C03636=1036.539,281.709,383.369,171.291,43.258,158.298
C03637=1036.532,281.461,383.400,171.287,43.257,158.298
C03638=1036.526,281.213,383.432,171.284,43.256,158.297
C03639=1036.519,280.965,383.463,171.280,43.255,158.297
C03640=1036.512,280.717,383.495,171.277,43.254,158.296
C03641=1036.506,280.468,383.525,171.273,43.253,158.295
C03642=1036.499,280.221,383.557,171.270,43.252,158.295
C03643=1036.492,279.973,383.588,171.266,43.251,158.294
C03644=1036.485,279.725,383.620,171.262,43.250,158.294
C03645=1036.479,279.477,383.651,171.259,43.249,158.293
C03646=1036.472,279.229,383.683,171.255,43.247,158.293
C03647=1036.465,278.981,383.714,171.252,43.247,158.292
C03648=1036.459,278.733,383.745,171.249,43.245,158.292
C03649=1036.452,278.485,383.776,171.245,43.244,158.291
C03650=1036.445,278.237,383.807,171.242,43.243,158.291
C03651=1036.438,277.989,383.838,171.238,43.242,158.290
C03652=1036.429,277.655,383.881,171.233,43.241,158.290
C03653=1036.420,277.319,383.922,171.229,43.240,158.289
C03654=1036.411,276.985,383.964,171.224,43.238,158.288
C03655=1036.401,276.651,384.006,171.219,43.237,158.288
C03656=1036.395,276.402,384.036,171.216,43.236,158.287
C03657=1036.388,276.154,384.068,171.212,43.235,158.287
C03658=1036.382,275.906,384.098,171.208,43.234,158.286
C03659=1036.374,275.658,384.129,171.205,43.233,158.286
C03660=1036.368,275.411,384.160,171.201,43.232,158.285
C03661=1036.362,275.162,384.191,171.198,43.231,158.285
C03662=1036.354,274.915,384.222,171.194,43.230,158.284
C03663=1036.348,274.666,384.253,171.191,43.229,158.284
C03664=1036.341,274.418,384.284,171.187,43.228,158.283
C03665=1036.335,274.170,384.315,171.185,43.227,158.283
C03666=1036.328,273.923,384.345,171.181,43.226,158.282
C03667=1036.321,273.674,384.376,171.177,43.225,158.282
C03668=1036.314,273.427,384.407,171.174,43.224,158.281
C03669=1036.308,273.178,384.438,171.170,43.223,158.281
C03670=1036.301,272.930,384.469,171.167,43.222,158.280
C03671=1036.294,272.682,384.499,171.163,43.222,158.280
C03672=1036.288,272.434,384.529,171.160,43.220,158.279
C03673=1036.280,272.187,384.560,171.156,43.220,158.279
C03674=1036.274,271.938,384.591,171.153,43.219,158.279
C03675=1036.267,271.690,384.622,171.150,43.217,158.278
C03676=1036.260,271.442,384.653,171.147,43.217,158.278
C03677=1036.254,271.194,384.683,171.143,43.216,158.277
C03678=1036.247,270.947,384.714,171.139,43.215,158.277
C03679=1036.240,270.698,384.744,171.136,43.214,158.276
C03680=1036.233,270.450,384.775,171.132,43.213,158.276
C03681=1036.227,270.202,384.805,171.129,43.212,158.275
C03682=1036.220,269.955,384.836,171.126,43.211,158.275
C03683=1036.214,269.706,384.866,171.123,43.210,158.274
C03684=1036.206,269.458,384.897,171.119,43.210,158.274
C03685=1036.201,269.210,384.927,171.116,43.208,158.273
C03686=1036.193,268.962,384.958,171.112,43.208,158.273
C03687=1036.187,268.714,384.989,171.109,43.207,158.272
C03688=1036.180,268.466,385.019,171.105,43.206,158.272
C03689=1036.173,268.218,385.048,171.103,43.205,158.272
C03690=1036.167,267.970,385.079,171.099,43.204,158.271
C03691=1036.159,267.721,385.109,171.096,43.203,158.271
C03692=1036.154,267.474,385.140,171.092,43.203,158.270
C03693=1036.146,267.225,385.170,171.089,43.202,158.270
C03694=1036.140,266.977,385.201,171.085,43.201,158.269
C03695=1036.133,266.730,385.231,171.083,43.200,158.269
C03696=1036.126,266.482,385.261,171.079,43.199,158.268
C03697=1036.120,266.233,385.292,171.076,43.198,158.268
C03698=1036.113,265.986,385.321,171.072,43.198,158.268
C03699=1036.106,265.737,385.352,171.069,43.197,158.267
C03700=1036.099,265.489,385.382,171.066,43.195,158.267
C03701=1036.093,265.241,385.412,171.063,43.195,158.266
C03702=1036.086,264.993,385.441,171.059,43.194,158.266
C03703=1036.079,264.744,385.472,171.056,43.193,158.265
C03704=1036.073,264.497,385.502,171.052,43.193,158.265
C03705=1036.066,264.248,385.532,171.050,43.192,158.265
C03706=1036.059,264.000,385.562,171.046,43.191,158.264
C03707=1036.052,263.753,385.592,171.043,43.190,158.264
C03708=1036.044,263.422,385.632,171.038,43.189,158.263
C03709=1036.035,263.092,385.672,171.035,43.188,158.263
C03710=1036.026,262.762,385.713,171.030,43.187,158.262
C03711=1036.017,262.432,385.752,171.025,43.185,158.261
C03712=1036.009,262.184,385.782,171.022,43.185,158.261
C03713=1036.004,261.935,385.812,171.019,43.184,158.260
C03714=1035.997,261.687,385.842,171.016,43.183,158.260
C03715=1035.990,261.440,385.872,171.012,43.182,158.260
C03716=1035.983,261.192,385.902,171.009,43.182,158.259
C03717=1035.976,260.943,385.931,171.006,43.181,158.259
C03718=1035.970,260.695,385.961,171.003,43.180,158.258
C03719=1035.963,260.446,385.991,171.000,43.179,158.258
C03720=1035.956,260.199,386.020,170.996,43.179,158.258
C03721=1035.948,259.951,386.050,170.993,43.179,158.257
C03722=1035.942,259.702,386.079,170.990,43.178,158.257
C03723=1035.935,259.455,386.109,170.987,43.177,158.256
C03724=1035.928,259.206,386.138,170.983,43.176,158.256
C03725=1035.922,258.958,386.168,170.980,43.176,158.256
C03726=1035.915,258.709,386.198,170.978,43.175,158.255
C03727=1035.908,258.462,386.227,170.974,43.174,158.255
C03728=1035.901,258.214,386.257,170.971,43.173,158.254
C03729=1035.894,257.965,386.287,170.967,43.173,158.254
C03730=1035.887,257.718,386.316,170.965,43.172,158.254
C03731=1035.880,257.469,386.345,170.961,43.172,158.253
C03732=1035.874,257.221,386.374,170.958,43.171,158.253
C03733=1035.867,256.972,386.405,170.955,43.170,158.252
C03734=1035.860,256.724,386.434,170.952,43.169,158.252
C03735=1035.853,256.476,386.464,170.949,43.169,158.252
C03736=1035.847,256.228,386.493,170.945,43.168,158.251
C03737=1035.840,255.980,386.523,170.943,43.167,158.251
C03738=1035.833,255.732,386.551,170.939,43.167,158.251
C03739=1035.826,255.483,386.581,170.936,43.166,158.250
C03740=1035.819,255.236,386.611,170.933,43.165,158.250
C03741=1035.813,254.987,386.640,170.930,43.165,158.249
C03742=1035.806,254.739,386.670,170.927,43.164,158.249
C03743=1035.800,254.491,386.699,170.923,43.163,158.248
C03744=1035.793,254.242,386.728,170.921,43.162,158.248
C03745=1035.786,253.995,386.757,170.917,43.162,158.248
C03746=1035.779,253.746,386.787,170.914,43.161,158.247
C03747=1035.772,253.498,386.816,170.912,43.161,158.247
C03748=1035.765,253.250,386.846,170.908,43.160,158.247
C03749=1035.759,253.002,386.875,170.905,43.159,158.246
C03750=1035.753,252.754,386.904,170.902,43.158,158.246
C03751=1035.746,252.505,386.933,170.899,43.158,158.245
C03752=1035.739,252.258,386.963,170.895,43.157,158.245
C03753=1035.732,252.009,386.992,170.893,43.157,158.245
C03754=1035.726,251.761,387.021,170.890,43.156,158.244
C03755=1035.719,251.513,387.050,170.886,43.155,158.244
C03756=1035.712,251.264,387.079,170.884,43.154,158.244
C03757=1035.706,251.016,387.109,170.880,43.154,158.243
C03758=1035.700,250.768,387.138,170.877,43.153,158.243
C03759=1035.692,250.520,387.167,170.874,43.153,158.242
C03760=1035.686,250.271,387.196,170.871,43.152,158.242
C03761=1035.680,250.023,387.225,170.869,43.151,158.242
C03762=1035.673,249.774,387.255,170.865,43.150,158.241
C03763=1035.666,249.527,387.284,170.862,43.149,158.241
C03764=1035.657,249.195,387.323,170.858,43.149,158.240
C03765=1035.648,248.864,387.362,170.854,43.148,158.240
C03766=1035.640,248.532,387.400,170.850,43.147,158.239
C03767=1035.631,248.201,387.440,170.846,43.146,158.239
C03768=1035.625,247.953,387.469,170.843,43.145,158.238
C03769=1035.618,247.705,387.498,170.840,43.145,158.238
C03770=1035.611,247.456,387.527,170.837,43.144,158.238
C03771=1035.604,247.208,387.556,170.834,43.144,158.237
C03772=1035.598,246.960,387.585,170.831,43.143,158.237
C03773=1035.592,246.712,387.614,170.828,43.142,158.237
C03774=1035.585,246.463,387.643,170.825,43.141,158.236
C03775=1035.579,246.215,387.672,170.822,43.140,158.236
C03776=1035.572,245.967,387.701,170.819,43.140,158.236
C03777=1035.566,245.719,387.730,170.816,43.139,158.235
C03778=1035.559,245.470,387.759,170.813,43.139,158.235
C03779=1035.553,245.222,387.788,170.811,43.138,158.234
C03780=1035.546,244.974,387.817,170.807,43.137,158.234
C03781=1035.539,244.726,387.846,170.805,43.137,158.234
C03782=1035.533,244.477,387.874,170.801,43.136,158.233
C03783=1035.527,244.228,387.903,170.798,43.135,158.233
C03784=1035.520,243.980,387.932,170.796,43.135,158.233
C03785=1035.513,243.732,387.961,170.792,43.134,158.232
C03786=1035.506,243.484,387.989,170.790,43.134,158.232
C03787=1035.500,243.235,388.018,170.786,43.133,158.232
C03788=1035.493,242.987,388.046,170.784,43.133,158.231
C03789=1035.487,242.739,388.075,170.781,43.132,158.231
C03790=1035.480,242.491,388.104,170.778,43.132,158.230
C03791=1035.474,242.243,388.132,170.775,43.131,158.230
C03792=1035.467,241.994,388.162,170.771,43.130,158.230
C03793=1035.460,241.746,388.190,170.769,43.130,158.229
C03794=1035.453,241.498,388.219,170.766,43.129,158.229
C03795=1035.447,241.249,388.247,170.763,43.128,158.229
C03796=1035.441,241.001,388.276,170.760,43.128,158.228
C03797=1035.434,240.753,388.304,170.758,43.127,158.228
C03798=1035.428,240.505,388.333,170.754,43.126,158.228
C03799=1035.420,240.256,388.361,170.752,43.126,158.227
C03800=1035.413,240.008,388.390,170.748,43.125,158.227
C03801=1035.407,239.759,388.418,170.746,43.125,158.227
C03802=1035.400,239.512,388.447,170.743,43.124,158.226
C03803=1035.393,239.263,388.474,170.740,43.124,158.226
C03804=1035.387,239.014,388.504,170.737,43.123,158.226
C03805=1035.380,238.766,388.532,170.735,43.123,158.225
C03806=1035.373,238.518,388.560,170.731,43.122,158.225
C03807=1035.366,238.270,388.588,170.729,43.122,158.225
C03808=1035.360,238.022,388.617,170.726,43.121,158.224
C03809=1035.353,237.773,388.644,170.723,43.121,158.224
C03810=1035.346,237.525,388.673,170.720,43.120,158.224
C03811=1035.340,237.277,388.701,170.718,43.120,158.223
C03812=1035.333,237.028,388.730,170.714,43.119,158.223
C03813=1035.326,236.780,388.758,170.712,43.119,158.223
C03814=1035.319,236.531,388.786,170.709,43.118,158.222
C03815=1035.312,236.283,388.814,170.706,43.118,158.222
C03816=1035.306,236.035,388.842,170.703,43.117,158.222
C03817=1035.300,235.787,388.871,170.700,43.117,158.221
C03818=1035.293,235.538,388.898,170.697,43.116,158.221
C03819=1035.286,235.290,388.926,170.695,43.116,158.221
C03820=1035.277,234.952,388.965,170.690,43.115,158.220
C03821=1035.269,234.615,389.003,170.687,43.114,158.220
C03822=1035.259,234.278,389.042,170.682,43.114,158.219
C03823=1035.250,233.940,389.080,170.679,43.113,158.219
C03824=1035.243,233.691,389.108,170.677,43.113,158.219
C03825=1035.236,233.444,389.136,170.673,43.112,158.218
C03826=1035.230,233.195,389.164,170.671,43.112,158.218
C03827=1035.223,232.947,389.192,170.667,43.111,158.218
C03828=1035.217,232.698,389.220,170.665,43.111,158.217
C03829=1035.210,232.450,389.248,170.662,43.110,158.217
C03830=1035.203,232.202,389.276,170.660,43.110,158.217
C03831=1035.197,231.953,389.304,170.657,43.109,158.216
C03832=1035.191,231.704,389.332,170.654,43.109,158.216
C03833=1035.184,231.457,389.361,170.651,43.108,158.216
C03834=1035.177,231.208,389.388,170.648,43.108,158.215
C03835=1035.170,230.960,389.416,170.646,43.107,158.215
C03836=1035.164,230.711,389.444,170.642,43.107,158.215
C03837=1035.157,230.463,389.472,170.640,43.106,158.214
C03838=1035.150,230.214,389.499,170.638,43.106,158.214
C03839=1035.144,229.966,389.527,170.635,43.105,158.214
C03840=1035.137,229.718,389.555,170.632,43.105,158.213
C03841=1035.130,229.470,389.583,170.629,43.104,158.213
C03842=1035.123,229.221,389.611,170.627,43.104,158.213
C03843=1035.117,228.974,389.638,170.624,43.103,158.213
C03844=1035.110,228.725,389.666,170.621,43.103,158.212
C03845=1035.104,228.477,389.694,170.618,43.102,158.212
C03846=1035.097,228.228,389.721,170.615,43.102,158.212
C03847=1035.090,227.980,389.749,170.613,43.101,158.211
C03848=1035.084,227.731,389.777,170.609,43.101,158.211
C03849=1035.077,227.483,389.805,170.607,43.101,158.211
C03850=1035.070,227.234,389.832,170.605,43.101,158.211
C03851=1035.064,226.986,389.860,170.602,43.100,158.210
C03852=1035.057,226.738,389.888,170.599,43.100,158.210
C03853=1035.050,226.489,389.915,170.596,43.099,158.210
C03854=1035.043,226.241,389.943,170.594,43.099,158.209
C03855=1035.037,225.992,389.970,170.591,43.098,158.209
C03856=1035.030,225.743,389.997,170.588,43.098,158.209
C03857=1035.023,225.495,390.025,170.586,43.097,158.208
C03858=1035.017,225.247,390.053,170.582,43.097,158.208
C03859=1035.009,224.998,390.080,170.580,43.097,158.208
C03860=1035.003,224.751,390.107,170.578,43.096,158.207
C03861=1034.996,224.502,390.135,170.575,43.096,158.207
C03862=1034.990,224.253,390.162,170.572,43.096,158.207
C03863=1034.983,224.005,390.190,170.570,43.095,158.207
C03864=1034.977,223.756,390.218,170.567,43.095,158.206
C03865=1034.969,223.508,390.245,170.564,43.094,158.206
C03866=1034.963,223.260,390.272,170.561,43.094,158.206
C03867=1034.956,223.011,390.299,170.559,43.093,158.205
C03868=1034.950,222.763,390.327,170.556,43.093,158.205
C03869=1034.943,222.515,390.355,170.553,43.093,158.205
C03870=1034.936,222.266,390.382,170.551,43.092,158.205
C03871=1034.930,222.017,390.409,170.549,43.092,158.204
C03872=1034.923,221.769,390.436,170.545,43.092,158.204
C03873=1034.916,221.520,390.464,170.543,43.091,158.204
C03874=1034.910,221.273,390.492,170.541,43.090,158.203
C03875=1034.903,221.024,390.518,170.537,43.090,158.203
C03876=1034.894,220.679,390.556,170.534,43.090,158.203
C03877=1034.885,220.334,390.594,170.530,43.089,158.202
C03878=1034.875,219.989,390.632,170.527,43.088,158.202
C03879=1034.866,219.644,390.670,170.523,43.087,158.201
C03880=1034.860,219.395,390.698,170.520,43.087,158.201
C03881=1034.853,219.148,390.724,170.518,43.087,158.201
C03882=1034.846,218.899,390.751,170.516,43.087,158.201
C03883=1034.839,218.651,390.779,170.513,43.087,158.200
C03884=1034.833,218.402,390.806,170.510,43.086,158.200
C03885=1034.825,218.154,390.833,170.508,43.085,158.200
C03886=1034.819,217.905,390.860,170.505,43.085,158.200
C03887=1034.812,217.657,390.887,170.502,43.085,158.199
C03888=1034.806,217.408,390.914,170.500,43.085,158.199
C03889=1034.798,217.160,390.941,170.497,43.084,158.199
C03890=1034.792,216.911,390.968,170.494,43.084,158.198
C03891=1034.786,216.663,390.995,170.492,43.083,158.198
C03892=1034.779,216.414,391.021,170.489,43.083,158.198
C03893=1034.772,216.166,391.049,170.487,43.083,158.198
C03894=1034.765,215.917,391.076,170.484,43.082,158.197
C03895=1034.759,215.669,391.103,170.481,43.082,158.197
C03896=1034.752,215.421,391.129,170.479,43.082,158.197
C03897=1034.745,215.172,391.156,170.477,43.081,158.197
C03898=1034.738,214.924,391.184,170.474,43.081,158.196
C03899=1034.732,214.675,391.210,170.471,43.080,158.196
C03900=1034.725,214.427,391.237,170.469,43.080,158.196
C03901=1034.718,214.178,391.264,170.466,43.080,158.196
C03902=1034.711,213.929,391.291,170.464,43.079,158.195
C03903=1034.705,213.681,391.318,170.461,43.079,158.195
C03904=1034.698,213.433,391.345,170.459,43.079,158.195
C03905=1034.692,213.184,391.372,170.456,43.078,158.194
C03906=1034.685,212.936,391.398,170.454,43.078,158.194
C03907=1034.678,212.687,391.425,170.451,43.078,158.194
C03908=1034.671,212.438,391.452,170.449,43.078,158.194
C03909=1034.665,212.191,391.479,170.446,43.077,158.193
C03910=1034.658,211.942,391.506,170.444,43.076,158.193
C03911=1034.652,211.693,391.533,170.441,43.076,158.193
C03912=1034.645,211.445,391.559,170.438,43.076,158.193
C03913=1034.639,211.196,391.586,170.436,43.076,158.192
C03914=1034.631,210.948,391.613,170.434,43.075,158.192
C03915=1034.625,210.700,391.639,170.430,43.075,158.192
C03916=1034.618,210.451,391.667,170.428,43.074,158.191
C03917=1034.611,210.202,391.693,170.426,43.074,158.191
C03918=1034.605,209.954,391.719,170.424,43.074,158.191
C03919=1034.598,209.705,391.746,170.420,43.074,158.191
C03920=1034.591,209.457,391.772,170.418,43.073,158.190
C03921=1034.585,209.208,391.799,170.416,43.073,158.190
C03922=1034.578,208.960,391.826,170.414,43.073,158.190
C03923=1034.571,208.712,391.852,170.411,43.072,158.190
C03924=1034.564,208.463,391.879,170.408,43.072,158.189
C03925=1034.558,208.214,391.906,170.406,43.071,158.189
C03926=1034.551,207.966,391.932,170.404,43.071,158.189
C03927=1034.544,207.717,391.958,170.401,43.071,158.189
C03928=1034.537,207.469,391.985,170.398,43.071,158.188
C03929=1034.531,207.220,392.011,170.396,43.071,158.188
C03930=1034.524,206.972,392.038,170.394,43.070,158.188
C03931=1034.518,206.723,392.064,170.391,43.070,158.188
C03932=1034.508,206.384,392.100,170.388,43.069,158.187
C03933=1034.498,206.045,392.136,170.385,43.069,158.187
C03934=1034.490,205.706,392.172,170.381,43.068,158.187
C03935=1034.481,205.366,392.208,170.378,43.068,158.186
C03936=1034.454,204.316,392.314,170.052,42.963,158.140
C03937=1034.448,204.068,392.339,170.048,42.964,158.140
C03938=1034.443,203.820,392.364,170.045,42.965,158.140
C03939=1034.436,203.571,392.389,170.042,42.965,158.140
C03940=1034.430,203.322,392.414,170.038,42.966,158.139
C03941=1034.424,203.073,392.439,170.034,42.966,158.139
C03942=1034.417,202.825,392.464,170.031,42.966,158.139
C03943=1034.412,202.577,392.489,170.027,42.967,158.139
C03944=1034.406,202.327,392.514,170.024,42.967,158.139
C03945=1034.400,202.079,392.539,170.021,42.968,158.139
C03946=1034.393,201.830,392.565,170.018,42.968,158.138
C03947=1034.388,201.581,392.589,170.014,42.969,158.138
C03948=1034.381,201.333,392.614,170.011,42.969,158.138
C03949=1034.375,201.084,392.639,170.008,42.970,158.138
C03950=1034.369,200.835,392.663,170.004,42.970,158.138
C03951=1034.363,200.587,392.689,170.001,42.971,158.138
C03952=1034.357,200.337,392.713,169.998,42.971,158.137
C03953=1034.351,200.090,392.738,169.994,42.972,158.137
C03954=1034.345,199.840,392.762,169.991,42.972,158.137
C03955=1034.338,199.592,392.787,169.987,42.973,158.137
C03956=1034.332,199.343,392.812,169.984,42.973,158.137
C03957=1034.325,199.094,392.837,169.980,42.974,158.137
C03958=1034.320,198.846,392.861,169.977,42.975,158.137
C03959=1034.313,198.597,392.886,169.974,42.975,158.137
C03960=1034.307,198.348,392.910,169.970,42.976,158.136
C03961=1034.300,198.099,392.934,169.967,42.977,158.136
C03962=1034.295,197.851,392.959,169.964,42.978,158.136
C03963=1034.288,197.602,392.983,169.960,42.978,158.136
C03964=1034.282,197.353,393.009,169.957,42.979,158.136
C03965=1034.275,197.104,393.033,169.954,42.979,158.136
C03966=1034.270,196.856,393.057,169.951,42.980,158.136
C03967=1034.263,196.608,393.082,169.947,42.980,158.136
C03968=1034.257,196.358,393.106,169.944,42.981,158.135
C03969=1034.252,196.110,393.130,169.941,42.981,158.135
C03970=1034.245,195.861,393.155,169.937,42.982,158.135
C03971=1034.239,195.612,393.180,169.934,42.983,158.135
C03972=1034.233,195.364,393.203,169.931,42.984,158.135
C03973=1034.227,195.115,393.229,169.928,42.984,158.135
C03974=1034.220,194.866,393.253,169.924,42.985,158.135
C03975=1034.215,194.617,393.277,169.921,42.985,158.135
C03976=1034.208,194.369,393.301,169.918,42.986,158.135
C03977=1034.202,194.120,393.326,169.915,42.986,158.134
C03978=1034.196,193.872,393.350,169.912,42.987,158.134
C03979=1034.190,193.622,393.375,169.908,42.988,158.134
C03980=1034.183,193.373,393.399,169.905,42.989,158.134
C03981=1034.178,193.125,393.423,169.902,42.989,158.134
C03982=1034.171,192.876,393.448,169.899,42.990,158.134
C03983=1034.166,192.628,393.472,169.895,42.991,158.134
C03984=1034.159,192.379,393.496,169.892,42.991,158.134
C03985=1034.153,192.129,393.521,169.889,42.992,158.133
C03986=1034.147,191.881,393.544,169.886,42.993,158.133
C03987=1034.141,191.632,393.569,169.883,42.993,158.133
C03988=1034.135,191.384,393.593,169.879,42.994,158.133
C03989=1034.128,191.135,393.617,169.876,42.994,158.133
C03990=1034.122,190.886,393.642,169.873,42.995,158.133
C03991=1034.116,190.638,393.666,169.870,42.995,158.133
C03992=1034.110,190.388,393.690,169.867,42.997,158.133
C03993=1034.104,190.140,393.714,169.864,42.997,158.133
C03994=1034.098,189.891,393.739,169.860,42.998,158.133
C03995=1034.092,189.643,393.762,169.857,42.998,158.132
C03996=1034.086,189.393,393.787,169.854,42.999,158.132
C03997=1034.080,189.110,393.815,169.850,43.000,158.132
C03998=1034.073,188.826,393.842,169.847,43.001,158.132
C03999=1034.066,188.541,393.870,169.843,43.001,158.132
C04000=1034.059,188.258,393.897,169.840,43.002,158.132
C04001=1034.053,188.010,393.921,169.837,43.002,158.132
C04002=1034.047,187.760,393.946,169.833,43.004,158.132
C04003=1034.041,187.512,393.969,169.830,43.004,158.132
C04004=1034.035,187.263,393.994,169.827,43.005,158.131
C04005=1034.029,187.015,394.018,169.824,43.005,158.131
C04006=1034.023,186.766,394.042,169.821,43.006,158.131
C04007=1034.017,186.517,394.066,169.818,43.007,158.131
C04008=1034.011,186.267,394.089,169.815,43.007,158.131
C04009=1034.006,186.019,394.113,169.812,43.008,158.131
C04010=1034.000,185.770,394.137,169.808,43.009,158.131
C04011=1033.994,185.521,394.162,169.805,43.010,158.131
C04012=1033.988,185.273,394.185,169.802,43.010,158.131
C04013=1033.982,185.024,394.210,169.799,43.011,158.131
C04014=1033.976,184.775,394.234,169.796,43.011,158.130
C04015=1033.970,184.527,394.258,169.793,43.012,158.130
C04016=1033.964,184.277,394.281,169.790,43.013,158.130
C04017=1033.958,184.029,394.305,169.787,43.013,158.130
C04018=1033.952,183.780,394.329,169.784,43.014,158.130
C04019=1033.946,183.531,394.353,169.781,43.015,158.130
C04020=1033.941,183.283,394.377,169.778,43.016,158.130
C04021=1033.935,183.033,394.401,169.774,43.016,158.130
C04022=1033.928,182.785,394.424,169.771,43.017,158.130
C04023=1033.922,182.536,394.448,169.768,43.018,158.130
C04024=1033.915,182.287,394.471,169.765,43.019,158.130
C04025=1033.909,182.038,394.495,169.762,43.020,158.130
C04026=1033.903,181.789,394.518,169.759,43.021,158.130
C04027=1033.897,181.541,394.541,169.756,43.022,158.130
C04028=1033.891,181.292,394.565,169.752,43.023,158.129
C04029=1033.885,181.043,394.588,169.750,43.024,158.129
C04030=1033.878,180.794,394.612,169.747,43.024,158.129
C04031=1033.872,180.545,394.635,169.744,43.025,158.129
C04032=1033.865,180.296,394.658,169.741,43.026,158.129
C04033=1033.859,180.048,394.682,169.738,43.027,158.129
C04034=1033.853,179.799,394.705,169.735,43.028,158.129
C04035=1033.847,179.550,394.729,169.731,43.029,158.129
C04036=1033.841,179.301,394.752,169.728,43.030,158.129
C04037=1033.834,179.052,394.776,169.725,43.031,158.129
C04038=1033.828,178.803,394.798,169.722,43.032,158.129
C04039=1033.822,178.555,394.822,169.719,43.033,158.129
C04040=1033.816,178.306,394.845,169.716,43.033,158.129
C04041=1033.810,178.057,394.869,169.714,43.035,158.129
C04042=1033.804,177.808,394.892,169.711,43.035,158.129
C04043=1033.797,177.559,394.915,169.708,43.036,158.129
C04044=1033.791,177.311,394.939,169.704,43.038,158.129
C04045=1033.785,177.062,394.961,169.701,43.038,158.129
C04046=1033.778,176.813,394.985,169.698,43.039,158.129
C04047=1033.773,176.564,395.008,169.695,43.040,158.129
C04048=1033.767,176.315,395.031,169.692,43.041,158.129
C04049=1033.760,176.066,395.055,169.689,43.042,158.129
C04050=1033.754,175.817,395.078,169.686,43.043,158.128
C04051=1033.748,175.569,395.100,169.683,43.044,158.129
C04052=1033.742,175.320,395.124,169.680,43.044,158.128
C04053=1033.736,175.071,395.147,169.678,43.045,158.128
C04054=1033.730,174.822,395.170,169.675,43.047,158.128
C04055=1033.724,174.573,395.193,169.672,43.047,158.128
C04056=1033.717,174.324,395.216,169.669,43.048,158.128
C04057=1033.711,174.076,395.239,169.666,43.049,158.128
C04058=1033.705,173.827,395.262,169.663,43.050,158.128
C04059=1033.699,173.578,395.286,169.660,43.051,158.128
C04060=1033.694,173.329,395.309,169.656,43.052,158.128
C04061=1033.687,173.068,395.333,169.653,43.053,158.128
C04062=1033.680,172.806,395.357,169.650,43.054,158.128
C04063=1033.673,172.545,395.382,169.647,43.055,158.128
C04064=1033.668,172.284,395.406,169.645,43.056,158.128
C04065=1033.662,172.035,395.428,169.642,43.057,158.128
C04066=1033.655,171.786,395.451,169.639,43.057,158.128
C04067=1033.649,171.537,395.475,169.636,43.059,158.128
C04068=1033.644,171.288,395.498,169.633,43.060,158.128
C04069=1033.638,171.040,395.521,169.630,43.060,158.128
C04070=1033.631,170.791,395.543,169.627,43.061,158.128
C04071=1033.625,170.541,395.567,169.624,43.063,158.128
C04072=1033.619,170.292,395.590,169.621,43.063,158.128
C04073=1033.614,170.044,395.613,169.618,43.064,158.128
C04074=1033.608,169.795,395.636,169.615,43.065,158.128
C04075=1033.601,169.547,395.659,169.613,43.066,158.128
C04076=1033.595,169.298,395.682,169.610,43.067,158.128
C04077=1033.590,169.049,395.705,169.607,43.068,158.127
C04078=1033.583,168.799,395.728,169.604,43.069,158.127
C04079=1033.578,168.550,395.751,169.601,43.070,158.128
C04080=1033.571,168.302,395.773,169.598,43.070,158.127
C04081=1033.565,168.053,395.796,169.595,43.072,158.127
C04082=1033.560,167.804,395.819,169.592,43.073,158.127
C04083=1033.554,167.555,395.842,169.589,43.073,158.127
C04084=1033.547,167.307,395.864,169.586,43.074,158.127
C04085=1033.542,167.058,395.887,169.584,43.076,158.127
C04086=1033.536,166.809,395.910,169.581,43.076,158.127
C04087=1033.530,166.560,395.933,169.578,43.077,158.127
C04088=1033.525,166.311,395.956,169.575,43.078,158.127
C04089=1033.517,166.062,395.979,169.572,43.079,158.127
C04090=1033.512,165.813,396.002,169.569,43.080,158.127
C04091=1033.506,165.564,396.025,169.566,43.081,158.127
C04092=1033.500,165.315,396.048,169.564,43.082,158.127
C04093=1033.494,165.066,396.070,169.561,43.083,158.127
C04094=1033.488,164.818,396.093,169.558,43.084,158.127
C04095=1033.482,164.569,396.116,169.555,43.085,158.127
C04096=1033.477,164.320,396.139,169.553,43.086,158.127
C04097=1033.470,164.071,396.161,169.550,43.087,158.127
C04098=1033.464,163.822,396.184,169.547,43.087,158.127
C04099=1033.459,163.573,396.206,169.544,43.089,158.127
C04100=1033.453,163.324,396.229,169.541,43.090,158.127
C04101=1033.447,163.052,396.254,169.538,43.090,158.127
C04102=1033.441,162.780,396.279,169.535,43.091,158.127
C04103=1033.434,162.509,396.304,169.532,43.093,158.127
C04104=1033.427,162.237,396.329,169.529,43.094,158.127
C04105=1033.422,161.987,396.351,169.526,43.094,158.127
C04106=1033.416,161.738,396.374,169.524,43.095,158.127
C04107=1033.410,161.489,396.397,169.521,43.097,158.127
C04108=1033.404,161.241,396.419,169.518,43.097,158.127
C04109=1033.398,160.993,396.442,169.515,43.098,158.127
C04110=1033.393,160.743,396.464,169.512,43.099,158.127
C04111=1033.387,160.494,396.486,169.510,43.100,158.127
C04112=1033.381,160.246,396.509,169.507,43.101,158.127
C04113=1033.375,159.997,396.532,169.504,43.102,158.127
C04114=1033.370,159.747,396.554,169.501,43.103,158.126
C04115=1033.363,159.499,396.577,169.498,43.104,158.126
C04116=1033.357,159.250,396.599,169.496,43.105,158.126
C04117=1033.351,159.000,396.621,169.493,43.106,158.126
C04118=1033.345,158.752,396.644,169.490,43.107,158.126
C04119=1033.339,158.503,396.665,169.487,43.108,158.126
C04120=1033.333,158.254,396.688,169.484,43.110,158.126
C04121=1033.327,158.005,396.711,169.481,43.111,158.127
C04122=1033.320,157.756,396.732,169.480,43.112,158.127
C04123=1033.315,157.507,396.755,169.477,43.113,158.127
C04124=1033.308,157.258,396.777,169.474,43.113,158.126
C04125=1033.302,156.973,396.803,169.470,43.115,158.126
C04126=1033.295,156.688,396.828,169.467,43.117,158.127
C04127=1033.288,156.404,396.853,169.464,43.118,158.127
C04128=1033.281,156.118,396.879,169.462,43.119,158.127
C04129=1033.274,155.869,396.901,169.459,43.119,158.126
C04130=1033.269,155.621,396.922,169.456,43.121,158.126
C04131=1033.262,155.372,396.945,169.453,43.122,158.127
C04132=1033.257,155.123,396.967,169.450,43.123,158.127
C04133=1033.251,154.874,396.989,169.447,43.124,158.127
C04134=1033.244,154.625,397.011,169.444,43.125,158.127
C04135=1033.239,154.376,397.034,169.442,43.126,158.127
C04136=1033.232,154.127,397.055,169.440,43.127,158.127
C04137=1033.226,153.878,397.077,169.437,43.129,158.127
C04138=1033.220,153.629,397.099,169.434,43.130,158.127
C04139=1033.214,153.380,397.122,169.431,43.131,158.127
C04140=1033.209,153.132,397.144,169.428,43.132,158.127
C04141=1033.202,152.883,397.165,169.426,43.133,158.127
C04142=1033.196,152.633,397.187,169.423,43.134,158.127
C04143=1033.190,152.385,397.209,169.420,43.136,158.127
C04144=1033.184,152.136,397.231,169.418,43.137,158.127
C04145=1033.178,151.886,397.253,169.415,43.138,158.127
C04146=1033.172,151.637,397.275,169.412,43.139,158.127
C04147=1033.166,151.389,397.297,169.410,43.140,158.127
C04148=1033.160,151.140,397.318,169.407,43.141,158.127
C04149=1033.154,150.891,397.340,169.404,43.142,158.127
C04150=1033.147,150.642,397.362,169.401,43.144,158.127
C04151=1033.142,150.392,397.384,169.399,43.144,158.127
C04152=1033.136,150.143,397.406,169.396,43.146,158.127
C04153=1033.130,149.895,397.427,169.394,43.147,158.127
C04154=1033.124,149.646,397.450,169.391,43.147,158.127
C04155=1033.118,149.397,397.471,169.388,43.149,158.127
C04156=1033.111,149.148,397.493,169.385,43.150,158.127
C04157=1033.105,148.899,397.515,169.383,43.151,158.127
C04158=1033.099,148.651,397.537,169.380,43.152,158.127
C04159=1033.093,148.401,397.558,169.378,43.154,158.127
C04160=1033.088,148.152,397.580,169.375,43.155,158.127
C04161=1033.082,147.903,397.602,169.372,43.156,158.127
C04162=1033.075,147.654,397.624,169.369,43.157,158.127
C04163=1033.070,147.405,397.645,169.367,43.158,158.127
C04164=1033.064,147.156,397.667,169.364,43.159,158.127
C04165=1033.057,146.907,397.689,169.362,43.161,158.127
C04166=1033.051,146.658,397.711,169.359,43.162,158.127
C04167=1033.045,146.409,397.732,169.356,43.163,158.127
C04168=1033.039,146.160,397.754,169.353,43.164,158.127
C04169=1033.033,145.911,397.775,169.351,43.165,158.127
C04170=1033.027,145.662,397.797,169.348,43.166,158.127
C04171=1033.020,145.413,397.818,169.346,43.167,158.127
C04172=1033.015,145.165,397.839,169.343,43.169,158.127
C04173=1033.008,144.915,397.861,169.340,43.170,158.127
C04174=1033.002,144.666,397.882,169.337,43.172,158.127
C04175=1032.996,144.417,397.904,169.336,43.173,158.128
C04176=1032.991,144.168,397.925,169.333,43.174,158.128
C04177=1032.984,143.919,397.947,169.330,43.175,158.128
C04178=1032.978,143.670,397.969,169.327,43.176,158.128
C04179=1032.972,143.421,397.990,169.324,43.177,158.128
C04180=1032.966,143.173,398.011,169.321,43.178,158.128
C04181=1032.960,142.923,398.033,169.320,43.179,158.128
C04182=1032.953,142.674,398.054,169.317,43.181,158.128
C04183=1032.947,142.425,398.076,169.314,43.182,158.128
C04184=1032.942,142.176,398.096,169.311,43.184,158.128
C04185=1032.936,141.927,398.118,169.308,43.185,158.128
C04186=1032.930,141.677,398.140,169.307,43.186,158.128
C04187=1032.924,141.429,398.161,169.304,43.187,158.128
C04188=1032.917,141.180,398.182,169.301,43.188,158.128
C04189=1032.911,140.895,398.207,169.298,43.189,158.128
C04190=1032.904,140.610,398.231,169.295,43.191,158.128
C04191=1032.897,140.325,398.256,169.293,43.192,158.128
C04192=1032.890,140.040,398.280,169.289,43.194,158.128
C04193=1032.884,139.791,398.302,169.287,43.195,158.128
C04194=1032.878,139.542,398.323,169.284,43.196,158.128
C04195=1032.872,139.292,398.344,169.281,43.197,158.128
C04196=1032.866,139.043,398.365,169.278,43.198,158.128
C04197=1032.860,138.795,398.386,169.277,43.200,158.128
C04198=1032.854,138.546,398.408,169.274,43.201,158.128
C04199=1032.848,138.296,398.429,169.271,43.202,158.128
C04200=1032.842,138.047,398.450,169.268,43.203,158.128
C04201=1032.835,137.798,398.471,169.265,43.204,158.128
C04202=1032.829,137.549,398.493,169.264,43.205,158.128
C04203=1032.824,137.300,398.513,169.261,43.207,158.129
C04204=1032.817,137.051,398.534,169.258,43.208,158.129
C04205=1032.811,136.802,398.556,169.255,43.210,158.129
C04206=1032.805,136.553,398.576,169.253,43.211,158.129
C04207=1032.799,136.304,398.597,169.251,43.212,158.129
C04208=1032.793,136.055,398.619,169.248,43.214,158.129
C04209=1032.787,135.806,398.640,169.245,43.215,158.129
C04210=1032.780,135.557,398.661,169.242,43.216,158.129
C04211=1032.775,135.308,398.682,169.241,43.217,158.129
C04212=1032.769,135.058,398.703,169.238,43.218,158.129
C04213=1032.763,134.810,398.723,169.235,43.220,158.129
C04214=1032.756,134.561,398.745,169.232,43.221,158.129
C04215=1032.750,134.311,398.765,169.230,43.222,158.129
C04216=1032.744,134.063,398.787,169.228,43.223,158.129
C04217=1032.738,133.813,398.808,169.225,43.224,158.129
C04218=1032.732,133.565,398.828,169.222,43.226,158.129
C04219=1032.726,133.315,398.849,169.220,43.227,158.129
C04220=1032.719,133.066,398.870,169.218,43.228,158.129
C04221=1032.714,132.818,398.892,169.215,43.230,158.129
C04222=1032.708,132.568,398.912,169.212,43.231,158.129
C04223=1032.702,132.320,398.933,169.210,43.232,158.130
C04224=1032.696,132.070,398.954,169.207,43.234,158.130
C04225=1032.689,131.822,398.975,169.205,43.235,158.130
C04226=1032.684,131.572,398.996,169.202,43.236,158.130
C04227=1032.678,131.323,399.017,169.200,43.237,158.130
C04228=1032.671,131.074,399.037,169.197,43.239,158.130
C04229=1032.666,130.825,399.058,169.194,43.240,158.130
C04230=1032.659,130.576,399.079,169.192,43.241,158.130
C04231=1032.653,130.327,399.100,169.190,43.242,158.130
C04232=1032.647,130.078,399.120,169.187,43.244,158.130
C04233=1032.641,129.828,399.141,169.184,43.245,158.130
C04234=1032.634,129.580,399.161,169.182,43.247,158.130
C04235=1032.628,129.330,399.182,169.180,43.248,158.130
C04236=1032.622,129.081,399.202,169.177,43.249,158.130
C04237=1032.615,128.833,399.223,169.174,43.251,158.130
C04238=1032.610,128.583,399.244,169.172,43.252,158.130
C04239=1032.604,128.334,399.264,169.169,43.253,158.130
C04240=1032.597,128.086,399.285,169.167,43.255,158.131
C04241=1032.591,127.836,399.305,169.164,43.256,158.131
C04242=1032.585,127.586,399.326,169.162,43.257,158.131
C04243=1032.579,127.338,399.347,169.159,43.259,158.131
C04244=1032.572,127.089,399.367,169.157,43.260,158.131
C04245=1032.567,126.840,399.388,169.154,43.262,158.131
C04246=1032.560,126.590,399.408,169.152,43.263,158.131
C04247=1032.554,126.342,399.429,169.149,43.264,158.131
C04248=1032.547,126.092,399.449,169.147,43.266,158.131
C04249=1032.542,125.843,399.470,169.144,43.267,158.131
C04250=1032.535,125.594,399.490,169.141,43.268,158.131
C04251=1032.529,125.345,399.511,169.139,43.270,158.131
C04252=1032.523,125.097,399.531,169.137,43.271,158.131
C04253=1032.516,124.811,399.554,169.134,43.272,158.131
C04254=1032.509,124.526,399.578,169.131,43.274,158.132
C04255=1032.502,124.241,399.601,169.128,43.276,158.132
C04256=1032.495,123.954,399.624,169.125,43.277,158.132
C04257=1032.489,123.706,399.645,169.122,43.279,158.132
C04258=1032.482,123.457,399.665,169.121,43.280,158.132
C04259=1032.476,123.208,399.685,169.118,43.281,158.132
C04260=1032.471,122.959,399.706,169.115,43.283,158.132
C04261=1032.465,122.709,399.726,169.113,43.284,158.132
C04262=1032.459,122.461,399.746,169.111,43.285,158.132
C04263=1032.452,122.212,399.767,169.108,43.287,158.132
C04264=1032.446,121.963,399.788,169.106,43.288,158.132
C04265=1032.440,121.713,399.808,169.103,43.289,158.132
C04266=1032.434,121.464,399.828,169.100,43.291,158.132
C04267=1032.428,121.215,399.848,169.098,43.292,158.133
C04268=1032.422,120.966,399.869,169.096,43.293,158.133
C04269=1032.416,120.717,399.889,169.093,43.295,158.133
C04270=1032.410,120.468,399.909,169.091,43.296,158.133
C04271=1032.403,120.218,399.929,169.089,43.298,158.133
C04272=1032.398,119.969,399.950,169.086,43.299,158.133
C04273=1032.392,119.720,399.970,169.083,43.301,158.133
C04274=1032.385,119.472,399.991,169.081,43.302,158.133
C04275=1032.379,119.223,400.011,169.079,43.303,158.133
C04276=1032.373,118.973,400.031,169.076,43.304,158.133
C04277=1032.367,118.724,400.052,169.074,43.306,158.133
C04278=1032.361,118.475,400.072,169.071,43.307,158.133
C04279=1032.355,118.226,400.092,169.068,43.308,158.133
C04280=1032.349,117.977,400.112,169.067,43.310,158.133
C04281=1032.344,117.728,400.132,169.064,43.311,158.133
C04282=1032.337,117.478,400.153,169.061,43.312,158.133
C04283=1032.331,117.230,400.173,169.060,43.314,158.134
C04284=1032.325,116.981,400.193,169.057,43.315,158.134
C04285=1032.319,116.731,400.214,169.054,43.316,158.134
C04286=1032.313,116.482,400.234,169.052,43.317,158.134
C04287=1032.307,116.233,400.253,169.049,43.319,158.134
C04288=1032.301,115.984,400.273,169.047,43.320,158.134
C04289=1032.295,115.734,400.293,169.045,43.321,158.134
C04290=1032.290,115.485,400.314,169.042,43.323,158.134
C04291=1032.284,115.236,400.334,169.039,43.324,158.134
C04292=1032.277,114.987,400.354,169.038,43.325,158.134
C04293=1032.271,114.738,400.374,169.035,43.326,158.134
C04294=1032.265,114.489,400.394,169.032,43.328,158.134
C04295=1032.260,114.240,400.414,169.030,43.329,158.134
C04296=1032.253,113.991,400.435,169.027,43.330,158.134
C04297=1032.247,113.742,400.455,169.026,43.331,158.134
C04298=1032.241,113.493,400.475,169.023,43.333,158.134
C04299=1032.236,113.243,400.494,169.020,43.334,158.134
C04300=1032.230,112.994,400.515,169.018,43.335,158.135
C04301=1032.224,112.745,400.535,169.016,43.337,158.135
C04302=1032.218,112.496,400.555,169.013,43.338,158.135
C04303=1032.211,112.247,400.575,169.011,43.339,158.135
C04304=1032.205,111.997,400.594,169.008,43.341,158.135
C04305=1032.199,111.749,400.614,169.006,43.342,158.135
C04306=1032.193,111.500,400.634,169.004,43.344,158.135
C04307=1032.186,111.250,400.654,169.001,43.345,158.135
C04308=1032.180,111.001,400.673,168.998,43.346,158.135
C04309=1032.174,110.752,400.693,168.997,43.348,158.135
C04310=1032.168,110.503,400.713,168.994,43.349,158.135
C04311=1032.162,110.253,400.733,168.991,43.351,158.135
C04312=1032.156,110.004,400.753,168.989,43.352,158.136
C04313=1032.150,109.755,400.773,168.987,43.354,158.136
C04314=1032.144,109.506,400.791,168.984,43.355,158.136
C04315=1032.137,109.257,400.812,168.982,43.357,158.136
C04316=1032.131,109.008,400.832,168.980,43.358,158.136
C04317=1032.124,108.723,400.853,168.977,43.360,158.136
C04318=1032.117,108.437,400.876,168.974,43.361,158.136
C04319=1032.110,108.151,400.899,168.971,43.363,158.136
C04320=1032.103,107.866,400.921,168.969,43.365,158.136
C04321=1032.097,107.617,400.941,168.966,43.366,158.136
C04322=1032.090,107.368,400.960,168.963,43.368,158.136
C04323=1032.084,107.119,400.980,168.962,43.369,158.137
C04324=1032.079,106.869,400.999,168.959,43.371,158.137
C04325=1032.073,106.621,401.019,168.956,43.372,158.137
C04326=1032.066,106.371,401.039,168.954,43.373,158.137
C04327=1032.060,106.122,401.058,168.952,43.375,158.137
C04328=1032.054,105.873,401.078,168.949,43.376,158.137
C04329=1032.048,105.624,401.097,168.947,43.377,158.137
C04330=1032.042,105.375,401.117,168.944,43.379,158.137
C04331=1032.035,105.126,401.136,168.942,43.380,158.137
C04332=1032.029,104.876,401.156,168.940,43.381,158.137
C04333=1032.023,104.627,401.175,168.937,43.383,158.137
C04334=1032.017,104.378,401.195,168.934,43.384,158.137
C04335=1032.011,104.129,401.214,168.933,43.386,158.138
C04336=1032.005,103.880,401.234,168.930,43.387,158.138
C04337=1031.999,103.631,401.253,168.927,43.389,158.138
C04338=1031.992,103.381,401.273,168.926,43.390,158.138
C04339=1031.986,103.132,401.292,168.923,43.391,158.138
C04340=1031.980,102.883,401.311,168.921,43.393,158.138
C04341=1031.974,102.634,401.331,168.918,43.394,158.138
C04342=1031.969,102.384,401.350,168.916,43.396,158.138
C04343=1031.962,102.136,401.370,168.914,43.397,158.138
C04344=1031.956,101.886,401.389,168.911,43.398,158.138
C04345=1031.950,101.638,401.409,168.908,43.400,158.138
C04346=1031.944,101.389,401.428,168.907,43.401,158.138
C04347=1031.938,101.138,401.447,168.904,43.403,158.139
C04348=1031.932,100.890,401.467,168.902,43.404,158.139
C04349=1031.926,100.640,401.486,168.899,43.405,158.139
C04350=1031.919,100.391,401.505,168.897,43.407,158.139
C04351=1031.913,100.142,401.525,168.895,43.408,158.139
C04352=1031.908,99.893,401.544,168.892,43.410,158.139
C04353=1031.901,99.644,401.563,168.889,43.411,158.139
C04354=1031.895,99.395,401.583,168.888,43.413,158.139
C04355=1031.889,99.146,401.602,168.885,43.414,158.139
C04356=1031.883,98.896,401.621,168.882,43.416,158.139
C04357=1031.876,98.646,401.640,168.881,43.417,158.139
C04358=1031.870,98.398,401.660,168.878,43.419,158.139
C04359=1031.864,98.149,401.678,168.875,43.420,158.139
C04360=1031.858,97.899,401.698,168.873,43.422,158.140
C04361=1031.852,97.650,401.716,168.871,43.423,158.140
C04362=1031.846,97.401,401.736,168.868,43.425,158.140
C04363=1031.839,97.152,401.755,168.866,43.426,158.140
C04364=1031.833,96.903,401.774,168.864,43.427,158.140
C04365=1031.827,96.653,401.793,168.862,43.429,158.140
C04366=1031.821,96.404,401.812,168.859,43.430,158.140
C04367=1031.815,96.155,401.831,168.857,43.432,158.140
C04368=1031.808,95.906,401.850,168.855,43.433,158.140
C04369=1031.803,95.657,401.869,168.852,43.435,158.141
C04370=1031.796,95.407,401.888,168.849,43.436,158.141
C04371=1031.790,95.158,401.908,168.848,43.438,158.141
C04372=1031.783,94.909,401.926,168.845,43.439,158.141
C04373=1031.778,94.659,401.946,168.842,43.441,158.141
C04374=1031.771,94.410,401.964,168.840,43.442,158.141
C04375=1031.765,94.162,401.984,168.838,43.444,158.141
C04376=1031.759,93.912,402.003,168.836,43.445,158.141
C04377=1031.753,93.663,402.021,168.833,43.447,158.141
C04378=1031.747,93.414,402.041,168.830,43.448,158.141
C04379=1031.740,93.164,402.059,168.829,43.450,158.141
C04380=1031.735,92.915,402.079,168.826,43.451,158.141
C04381=1031.728,92.630,402.101,168.823,43.453,158.142
C04382=1031.721,92.345,402.121,168.821,43.454,158.142
C04383=1031.713,92.059,402.144,168.818,43.456,158.142
C04384=1031.707,91.773,402.165,168.815,43.457,158.142
C04385=1031.701,91.524,402.184,168.812,43.459,158.142
C04386=1031.695,91.275,402.203,168.811,43.460,158.142
C04387=1031.689,91.025,402.222,168.808,43.462,158.142
C04388=1031.682,90.776,402.241,168.806,43.463,158.142
C04389=1031.676,90.527,402.259,168.804,43.464,158.142
C04390=1031.670,90.278,402.278,168.801,43.466,158.142
C04391=1031.664,90.029,402.297,168.799,43.467,158.142
C04392=1031.658,89.779,402.316,168.797,43.469,158.143
C04393=1031.652,89.530,402.335,168.795,43.470,158.143
C04394=1031.645,89.281,402.354,168.792,43.472,158.143
C04395=1031.639,89.032,402.372,168.789,43.474,158.143
C04396=1031.632,88.783,402.391,168.788,43.475,158.143
C04397=1031.627,88.534,402.409,168.785,43.477,158.143
C04398=1031.621,88.285,402.428,168.782,43.478,158.143
C04399=1031.615,88.036,402.447,168.781,43.480,158.143
C04400=1031.608,87.786,402.465,168.778,43.481,158.143
C04401=1031.602,87.537,402.484,168.775,43.483,158.143
C04402=1031.596,87.288,402.502,168.774,43.484,158.144
C04403=1031.589,87.039,402.521,168.771,43.486,158.144
C04404=1031.583,86.789,402.540,168.768,43.487,158.144
C04405=1031.577,86.540,402.559,168.766,43.489,158.144
C04406=1031.571,86.290,402.577,168.764,43.490,158.144
C04407=1031.564,86.041,402.595,168.762,43.492,158.144
C04408=1031.558,85.792,402.614,168.759,43.493,158.144
C04409=1031.552,85.543,402.633,168.757,43.495,158.144
C04410=1031.545,85.294,402.651,168.755,43.496,158.144
C04411=1031.539,85.044,402.669,168.752,43.498,158.145
C04412=1031.534,84.795,402.688,168.750,43.500,158.145
C04413=1031.528,84.546,402.707,168.748,43.501,158.145
C04414=1031.521,84.297,402.726,168.745,43.503,158.145
C04415=1031.515,84.047,402.743,168.742,43.504,158.145
C04416=1031.509,83.798,402.762,168.741,43.505,158.145
C04417=1031.502,83.549,402.781,168.738,43.507,158.145
C04418=1031.496,83.300,402.799,168.736,43.508,158.145
C04419=1031.490,83.050,402.818,168.734,43.510,158.145
C04420=1031.485,82.802,402.836,168.731,43.511,158.145
C04421=1031.478,82.552,402.855,168.729,43.513,158.146
C04422=1031.472,82.303,402.873,168.726,43.514,158.146
C04423=1031.466,82.054,402.891,168.725,43.516,158.146
C04424=1031.459,81.804,402.910,168.722,43.517,158.146
C04425=1031.453,81.555,402.929,168.719,43.519,158.146
C04426=1031.447,81.306,402.947,168.717,43.520,158.146
C04427=1031.441,81.057,402.965,168.715,43.522,158.146
C04428=1031.435,80.808,402.984,168.712,43.523,158.146
C04429=1031.429,80.558,403.002,168.710,43.525,158.146
C04430=1031.423,80.309,403.021,168.708,43.526,158.146
C04431=1031.416,80.059,403.039,168.706,43.528,158.146
C04432=1031.411,79.811,403.057,168.703,43.529,158.146
C04433=1031.404,79.562,403.076,168.700,43.531,158.147
C04434=1031.398,79.312,403.094,168.699,43.532,158.147
C04435=1031.392,79.063,403.112,168.696,43.534,158.147
C04436=1031.385,78.814,403.131,168.694,43.535,158.147
C04437=1031.380,78.564,403.149,168.692,43.536,158.147
C04438=1031.374,78.315,403.168,168.689,43.538,158.147
C04439=1031.368,78.065,403.186,168.687,43.539,158.147
C04440=1031.361,77.816,403.204,168.685,43.541,158.147
C04441=1031.355,77.566,403.222,168.683,43.542,158.147
C04442=1031.349,77.318,403.241,168.680,43.544,158.147
C04443=1031.343,77.068,403.258,168.677,43.545,158.147
C04444=1031.337,76.819,403.277,168.676,43.547,158.148
C04445=1031.330,76.534,403.298,168.673,43.549,158.148
C04446=1031.322,76.249,403.318,168.670,43.551,158.148
C04447=1031.315,75.963,403.339,168.668,43.552,158.148
C04448=1031.308,75.677,403.359,168.665,43.554,158.148
C04449=1031.302,75.428,403.378,168.662,43.556,158.148
C04450=1031.296,75.179,403.396,168.659,43.557,158.148
C04451=1031.289,74.929,403.414,168.658,43.559,158.148
C04452=1031.284,74.680,403.432,168.655,43.560,158.149
C04453=1031.278,74.431,403.450,168.653,43.561,158.149
C04454=1031.271,74.181,403.468,168.651,43.563,158.149
C04455=1031.264,73.932,403.486,168.648,43.565,158.149
C04456=1031.258,73.684,403.504,168.646,43.566,158.149
C04457=1031.252,73.434,403.522,168.644,43.568,158.149
C04458=1031.246,73.184,403.540,168.641,43.569,158.149
C04459=1031.240,72.935,403.559,168.639,43.571,158.149
C04460=1031.234,72.686,403.576,168.637,43.573,158.149
C04461=1031.227,72.437,403.593,168.635,43.574,158.149
C04462=1031.221,72.187,403.612,168.632,43.576,158.150
C04463=1031.215,71.938,403.630,168.629,43.577,158.150
C04464=1031.209,71.689,403.648,168.628,43.579,158.150
C04465=1031.203,71.440,403.666,168.625,43.580,158.150
C04466=1031.196,71.190,403.684,168.622,43.582,158.150
C04467=1031.191,70.941,403.701,168.621,43.583,158.150
C04468=1031.184,70.692,403.720,168.618,43.585,158.150
C04469=1031.178,70.442,403.738,168.616,43.586,158.150
C04470=1031.172,70.193,403.755,168.614,43.587,158.150
C04471=1031.165,69.944,403.773,168.611,43.589,158.150
C04472=1031.159,69.695,403.791,168.609,43.591,158.151
C04473=1031.154,69.446,403.809,168.606,43.592,158.151
C04474=1031.148,69.196,403.827,168.604,43.594,158.151
C04475=1031.141,68.947,403.845,168.602,43.595,158.151
C04476=1031.134,68.697,403.863,168.599,43.597,158.151
C04477=1031.129,68.448,403.880,168.598,43.599,158.151
C04478=1031.122,68.199,403.898,168.595,43.600,158.151
C04479=1031.116,67.949,403.916,168.592,43.602,158.151
C04480=1031.110,67.700,403.933,168.591,43.603,158.151
C04481=1031.103,67.451,403.951,168.588,43.605,158.151
C04482=1031.097,67.201,403.969,168.585,43.606,158.152
C04483=1031.091,66.952,403.987,168.583,43.607,158.152
C04484=1031.085,66.703,404.004,168.581,43.609,158.152
C04485=1031.078,66.453,404.022,168.579,43.611,158.152
C04486=1031.073,66.204,404.040,168.576,43.612,158.152
C04487=1031.066,65.955,404.057,168.574,43.614,158.152
C04488=1031.060,65.706,404.075,168.572,43.616,158.152
C04489=1031.053,65.457,404.093,168.569,43.617,158.152
C04490=1031.047,65.207,404.110,168.567,43.619,158.152
C04491=1031.042,64.958,404.128,168.565,43.620,158.152
C04492=1031.035,64.709,404.145,168.562,43.622,158.153
C04493=1031.029,64.459,404.163,168.560,43.624,158.153
C04494=1031.023,64.210,404.180,168.558,43.625,158.153
C04495=1031.016,63.961,404.198,168.555,43.627,158.153
C04496=1031.011,63.711,404.216,168.554,43.628,158.153
C04497=1031.004,63.462,404.233,168.551,43.629,158.153
C04498=1030.997,63.213,404.250,168.548,43.631,158.153
C04499=1030.992,62.964,404.268,168.547,43.633,158.153
C04500=1030.985,62.714,404.285,168.544,43.635,158.153
C04501=1030.978,62.465,404.303,168.541,43.636,158.153
C04502=1030.972,62.216,404.320,168.539,43.638,158.154
C04503=1030.966,61.966,404.338,168.537,43.640,158.154
C04504=1030.959,61.718,404.355,168.534,43.642,158.154
C04505=1030.953,61.467,404.372,168.531,43.643,158.154
C04506=1030.947,61.218,404.389,168.530,43.644,158.154
C04507=1030.940,60.969,404.406,168.527,43.646,158.154
C04508=1030.934,60.719,404.424,168.525,43.648,158.154
C04509=1030.927,60.434,404.443,168.522,43.650,158.155
C04510=1030.920,60.148,404.463,168.519,43.652,158.155
C04511=1030.912,59.863,404.483,168.517,43.654,158.155
C04512=1030.905,59.577,404.503,168.514,43.656,158.155
C04513=1030.899,59.327,404.520,168.511,43.657,158.155
C04514=1030.893,59.078,404.538,168.510,43.659,158.155
C04515=1030.886,58.829,404.555,168.507,43.660,158.155
C04516=1030.879,58.580,404.572,168.504,43.662,158.155
C04517=1030.873,58.330,404.589,168.503,43.663,158.155
C04518=1030.867,58.081,404.607,168.500,43.665,158.156
C04519=1030.861,57.831,404.623,168.497,43.667,158.156
C04520=1030.854,57.582,404.640,168.496,43.668,158.156
C04521=1030.848,57.333,404.658,168.493,43.670,158.156
C04522=1030.842,57.084,404.675,168.490,43.672,158.156
C04523=1030.835,56.834,404.693,168.489,43.674,158.156
C04524=1030.829,56.585,404.709,168.486,43.675,158.156
C04525=1030.823,56.335,404.727,168.483,43.677,158.156
C04526=1030.817,56.087,404.744,168.482,43.678,158.157
C04527=1030.810,55.837,404.761,168.479,43.680,158.157
C04528=1030.805,55.587,404.778,168.476,43.681,158.157
C04529=1030.798,55.338,404.795,168.475,43.683,158.157
C04530=1030.791,55.089,404.812,168.472,43.685,158.157
C04531=1030.785,54.839,404.829,168.469,43.686,158.157
C04532=1030.779,54.590,404.846,168.468,43.688,158.157
C04533=1030.773,54.341,404.864,168.465,43.690,158.157
C04534=1030.766,54.092,404.881,168.462,43.691,158.157
C04535=1030.760,53.842,404.898,168.461,43.693,158.157
C04536=1030.754,53.593,404.915,168.458,43.695,158.158
C04537=1030.747,53.344,404.932,168.455,43.696,158.158
C04538=1030.741,53.094,404.949,168.453,43.697,158.158
C04539=1030.735,52.844,404.966,168.451,43.699,158.158
C04540=1030.729,52.596,404.983,168.448,43.701,158.158
C04541=1030.723,52.346,405.000,168.446,43.702,158.158
C04542=1030.716,52.097,405.017,168.444,43.704,158.158
C04543=1030.711,51.848,405.035,168.442,43.705,158.158
C04544=1030.704,51.598,405.051,168.439,43.707,158.158
C04545=1030.698,51.349,405.068,168.437,43.708,158.158
C04546=1030.691,51.099,405.085,168.435,43.710,158.159
C04547=1030.686,50.850,405.102,168.432,43.712,158.159
C04548=1030.680,50.601,405.119,168.429,43.713,158.159
C04549=1030.673,50.351,405.136,168.428,43.715,158.159
C04550=1030.667,50.103,405.153,168.425,43.717,158.159
C04551=1030.661,49.852,405.170,168.422,43.718,158.159
C04552=1030.655,49.603,405.187,168.421,43.720,158.159
C04553=1030.648,49.355,405.204,168.418,43.721,158.159
C04554=1030.642,49.105,405.221,168.415,43.723,158.159
C04555=1030.636,48.856,405.238,168.414,43.724,158.160
C04556=1030.630,48.606,405.255,168.411,43.726,158.159
C04557=1030.624,48.357,405.272,168.409,43.727,158.160
C04558=1030.618,48.107,405.288,168.407,43.728,158.160
C04559=1030.611,47.858,405.306,168.404,43.730,158.160
C04560=1030.606,47.608,405.322,168.402,43.732,158.160
C04561=1030.599,47.360,405.339,168.399,43.733,158.160
C04562=1030.593,47.110,405.356,168.397,43.735,158.160
C04563=1030.587,46.861,405.374,168.395,43.736,158.160
C04564=1030.581,46.611,405.390,168.392,43.738,158.160
C04565=1030.574,46.362,405.407,168.390,43.740,158.160
C04566=1030.568,46.112,405.423,168.388,43.741,158.160
C04567=1030.563,45.863,405.441,168.385,43.743,158.161
C04568=1030.556,45.613,405.458,168.384,43.744,158.161
C04569=1030.550,45.365,405.475,168.381,43.746,158.161
C04570=1030.544,45.115,405.491,168.378,43.747,158.161
C04571=1030.538,44.866,405.509,168.376,43.749,158.161
C04572=1030.532,44.616,405.525,168.374,43.750,158.161
C04573=1030.524,44.331,405.544,168.371,43.752,158.161
C04574=1030.518,44.045,405.563,168.368,43.754,158.161
C04575=1030.511,43.759,405.583,168.366,43.756,158.161
C04576=1030.504,43.473,405.602,168.363,43.757,158.161
C04577=1030.498,43.223,405.618,168.360,43.759,158.161
C04578=1030.492,42.973,405.636,168.359,43.760,158.162
C04579=1030.486,42.724,405.652,168.356,43.762,158.162
C04580=1030.480,42.475,405.669,168.353,43.763,158.162
C04581=1030.473,42.225,405.686,168.352,43.765,158.162
C04582=1030.467,41.976,405.702,168.349,43.766,158.162
C04583=1030.461,41.727,405.718,168.346,43.768,158.162
C04584=1030.454,41.477,405.734,168.345,43.770,158.162
C04585=1030.448,41.228,405.751,168.342,43.771,158.162
C04586=1030.442,40.979,405.768,168.339,43.773,158.162
C04587=1030.436,40.729,405.784,168.338,43.775,158.163
C04588=1030.429,40.479,405.800,168.335,43.776,158.163
C04589=1030.423,40.231,405.817,168.332,43.778,158.163
C04590=1030.417,39.981,405.834,168.331,43.780,158.163
C04591=1030.411,39.732,405.850,168.328,43.781,158.163
C04592=1030.405,39.482,405.867,168.325,43.783,158.163
C04593=1030.398,39.233,405.884,168.324,43.784,158.163
C04594=1030.392,38.984,405.900,168.321,43.786,158.163
C04595=1030.386,38.735,405.916,168.318,43.787,158.163
C04596=1030.380,38.484,405.933,168.316,43.789,158.163
C04597=1030.374,38.235,405.949,168.314,43.790,158.163
C04598=1030.368,37.986,405.966,168.311,43.792,158.164
C04599=1030.362,37.737,405.982,168.308,43.794,158.164
C04600=1030.355,37.487,405.999,168.307,43.795,158.164
C04601=1030.349,37.238,406.015,168.304,43.797,158.164
C04602=1030.342,36.989,406.031,168.301,43.799,158.164
C04603=1030.337,36.739,406.047,168.300,43.800,158.164
C04604=1030.330,36.489,406.064,168.297,43.802,158.164
C04605=1030.324,36.240,406.080,168.294,43.804,158.164
C04606=1030.317,35.991,406.096,168.293,43.805,158.164
C04607=1030.311,35.741,406.112,168.290,43.807,158.164
C04608=1030.305,35.492,406.128,168.287,43.809,158.165
C04609=1030.299,35.242,406.145,168.285,43.810,158.165
C04610=1030.292,34.993,406.160,168.283,43.812,158.165
C04611=1030.286,34.744,406.177,168.280,43.813,158.165
C04612=1030.280,34.494,406.193,168.278,43.815,158.165
C04613=1030.274,34.245,406.209,168.276,43.817,158.165
C04614=1030.267,33.995,406.225,168.273,43.819,158.165
C04615=1030.261,33.746,406.241,168.271,43.820,158.165
C04616=1030.255,33.497,406.258,168.268,43.822,158.165
C04617=1030.248,33.248,406.273,168.266,43.824,158.166
C04618=1030.243,32.998,406.290,168.263,43.825,158.166
C04619=1030.236,32.748,406.306,168.261,43.827,158.166
C04620=1030.229,32.499,406.322,168.259,43.829,158.166
C04621=1030.223,32.250,406.338,168.257,43.830,158.166
C04622=1030.217,32.000,406.354,168.254,43.832,158.166
C04623=1030.211,31.751,406.370,168.251,43.834,158.166
C04624=1030.205,31.502,406.386,168.250,43.835,158.166
C04625=1030.199,31.253,406.403,168.247,43.836,158.166
C04626=1030.192,31.003,406.419,168.244,43.838,158.166
C04627=1030.186,30.754,406.435,168.243,43.840,158.167
C04628=1030.180,30.504,406.451,168.240,43.841,158.167
C04629=1030.174,30.255,406.467,168.237,43.843,158.167
C04630=1030.167,30.005,406.482,168.234,43.845,158.167
C04631=1030.161,29.756,406.499,168.233,43.847,158.167
C04632=1030.155,29.507,406.515,168.230,43.848,158.167
C04633=1030.149,29.257,406.530,168.227,43.850,158.167
C04634=1030.143,29.008,406.547,168.226,43.852,158.167
C04635=1030.136,28.758,406.563,168.223,43.853,158.167
C04636=1030.129,28.509,406.579,168.220,43.855,158.167
C04637=1030.123,28.223,406.597,168.218,43.857,158.168
C04638=1030.116,27.937,406.615,168.215,43.859,158.168
C04639=1030.109,27.651,406.633,168.213,43.860,158.168
C04640=1030.101,27.365,406.652,168.210,43.862,158.168
C04641=1030.095,27.115,406.667,168.207,43.864,158.168
C04642=1030.089,26.866,406.683,168.204,43.865,158.168
C04643=1030.082,26.617,406.699,168.202,43.867,158.168
C04644=1030.076,26.367,406.715,168.200,43.869,158.168
C04645=1030.070,26.118,406.730,168.197,43.870,158.168
C04646=1030.064,25.868,406.746,168.195,43.872,158.169
C04647=1030.057,25.619,406.762,168.192,43.874,158.169
C04648=1030.051,25.369,406.778,168.191,43.876,158.169
C04649=1030.044,25.120,406.794,168.188,43.878,158.169
C04650=1030.038,24.870,406.810,168.185,43.879,158.169
C04651=1030.032,24.621,406.825,168.183,43.881,158.169
C04652=1030.026,24.371,406.841,168.181,43.883,158.169
C04653=1030.019,24.122,406.857,168.178,43.884,158.169
C04654=1030.014,23.872,406.872,168.175,43.886,158.169
C04655=1030.007,23.623,406.888,168.173,43.888,158.169
C04656=1030.000,23.374,406.904,168.171,43.889,158.170
C04657=1029.995,23.124,406.919,168.169,43.891,158.170
C04658=1029.988,22.875,406.935,168.166,43.892,158.170
C04659=1029.982,22.625,406.950,168.163,43.894,158.170
C04660=1029.976,22.376,406.966,168.162,43.896,158.170
C04661=1029.970,22.127,406.982,168.159,43.897,158.170
C04662=1029.963,21.877,406.997,168.156,43.899,158.170
C04663=1029.957,21.628,407.014,168.154,43.901,158.170
C04664=1029.951,21.378,407.028,168.152,43.903,158.171
C04665=1029.944,21.129,407.044,168.149,43.904,158.170
C04666=1029.939,20.879,407.060,168.147,43.906,158.171
C04667=1029.932,20.630,407.075,168.144,43.908,158.171
C04668=1029.926,20.381,407.092,168.142,43.909,158.171
C04669=1029.920,20.131,407.107,168.139,43.911,158.171
C04670=1029.914,19.882,407.123,168.137,43.913,158.171
C04671=1029.907,19.632,407.138,168.134,43.914,158.171
C04672=1029.901,19.383,407.153,168.132,43.916,158.171
C04673=1029.895,19.133,407.169,168.130,43.917,158.171
C04674=1029.889,18.884,407.184,168.127,43.919,158.171
C04675=1029.882,18.635,407.200,168.125,43.921,158.172
C04676=1029.876,18.385,407.215,168.122,43.922,158.172
C04677=1029.870,18.136,407.231,168.120,43.924,158.172
C04678=1029.863,17.886,407.246,168.118,43.926,158.172
C04679=1029.857,17.637,407.261,168.115,43.928,158.172
C04680=1029.852,17.388,407.277,168.112,43.930,158.172
C04681=1029.845,17.138,407.291,168.110,43.931,158.172
C04682=1029.838,16.889,407.307,168.108,43.933,158.172
C04683=1029.833,16.639,407.323,168.105,43.935,158.172
C04684=1029.826,16.390,407.338,168.103,43.937,158.173
C04685=1029.820,16.140,407.353,168.100,43.938,158.173
C04686=1029.813,15.891,407.368,168.098,43.940,158.173
C04687=1029.807,15.641,407.384,168.096,43.941,158.173
C04688=1029.801,15.392,407.399,168.093,43.943,158.173
C04689=1029.795,15.142,407.414,168.090,43.945,158.173
C04690=1029.789,14.893,407.431,168.088,43.947,158.173
C04691=1029.783,14.644,407.445,168.086,43.948,158.173
C04692=1029.777,14.394,407.460,168.083,43.949,158.173
C04693=1029.770,14.145,407.476,168.080,43.951,158.173
C04694=1029.764,13.895,407.491,168.078,43.953,158.173
C04695=1029.758,13.645,407.506,168.076,43.955,158.174
C04696=1029.751,13.396,407.521,168.073,43.956,158.174
C04697=1029.745,13.147,407.537,168.071,43.958,158.174
C04698=1029.738,12.897,407.552,168.068,43.960,158.174
C04699=1029.732,12.647,407.567,168.066,43.962,158.174
C04700=1029.726,12.398,407.582,168.063,43.964,158.174
C04701=1029.719,12.113,407.599,168.060,43.966,158.174
C04702=1029.711,11.829,407.616,168.058,43.968,158.174
C04703=1029.704,11.544,407.633,168.055,43.970,158.174
C04704=1029.697,11.259,407.651,168.052,43.972,158.175
C04705=1029.690,11.010,407.666,168.050,43.973,158.175
C04706=1029.684,10.760,407.681,168.047,43.975,158.175
C04707=1029.678,10.511,407.695,168.045,43.977,158.175
C04708=1029.672,10.261,407.710,168.042,43.979,158.175
C04709=1029.665,10.012,407.725,168.039,43.981,158.175
C04710=1029.659,9.762,407.740,168.037,43.983,158.175
C04711=1029.652,9.512,407.755,168.034,43.984,158.175
C04712=1029.646,9.263,407.771,168.032,43.986,158.176
C04713=1029.640,9.014,407.785,168.030,43.988,158.176
C04714=1029.634,8.765,407.800,168.027,43.990,158.176
C04715=1029.627,8.515,407.815,168.025,43.992,158.176
C04716=1029.621,8.265,407.830,168.022,43.993,158.176
C04717=1029.614,8.016,407.845,168.019,43.995,158.176
C04718=1029.609,7.767,407.860,168.018,43.996,158.176
C04719=1029.602,7.517,407.875,168.015,43.998,158.176
C04720=1029.596,7.267,407.890,168.012,44.000,158.176
C04721=1029.590,7.018,407.904,168.010,44.002,158.177
C04722=1029.583,6.768,407.919,168.007,44.003,158.176
C04723=1029.577,6.519,407.934,168.004,44.005,158.177
C04724=1029.571,6.269,407.949,168.003,44.007,158.177
C04725=1029.565,6.020,407.964,168.000,44.009,158.177
C04726=1029.558,5.770,407.979,167.997,44.011,158.177
C04727=1029.552,5.521,407.993,167.995,44.012,158.177
C04728=1029.546,5.272,408.008,167.992,44.014,158.177
C04729=1029.540,5.022,408.023,167.989,44.016,158.177
C04730=1029.533,4.772,408.038,167.987,44.018,158.177
C04731=1029.527,4.523,408.053,167.985,44.020,158.178
C04732=1029.521,4.274,408.068,167.982,44.021,158.178
C04733=1029.515,4.024,408.083,167.980,44.023,158.178
C04734=1029.509,3.775,408.097,167.977,44.025,158.178
C04735=1029.503,3.525,408.112,167.974,44.026,158.178
C04736=1029.496,3.276,408.127,167.972,44.028,158.178
C04737=1029.490,3.026,408.142,167.970,44.029,158.178
C04738=1029.483,2.777,408.156,167.967,44.031,158.178
C04739=1029.477,2.527,408.170,167.965,44.033,158.178
C04740=1029.471,2.277,408.185,167.962,44.035,158.178
C04741=1029.465,2.028,408.200,167.959,44.036,158.178
C04742=1029.459,1.779,408.215,167.957,44.038,158.179
C04743=1029.452,1.529,408.230,167.955,44.040,158.179
C04744=1029.446,1.280,408.244,167.952,44.041,158.179
C04745=1029.440,1.031,408.259,167.950,44.043,158.179
C04746=1029.434,0.781,408.274,167.947,44.045,158.179
C04747=1029.428,0.531,408.288,167.945,44.047,158.179
C04748=1029.422,0.282,408.303,167.942,44.048,158.179
C04749=1029.415,0.032,408.318,167.940,44.050,158.179
C04750=1029.410,-0.217,408.333,167.937,44.052,158.179
C04751=1029.403,-0.467,408.348,167.935,44.053,158.179
C04752=1029.398,-0.716,408.362,167.932,44.055,158.179
C04753=1029.391,-0.966,408.376,167.929,44.057,158.180
C04754=1029.385,-1.215,408.391,167.927,44.059,158.180
C04755=1029.379,-1.464,408.406,167.924,44.060,158.180
C04756=1029.373,-1.714,408.421,167.922,44.062,158.180
C04757=1029.367,-1.964,408.435,167.920,44.064,158.180
C04758=1029.360,-2.213,408.449,167.917,44.065,158.180
C04759=1029.354,-2.463,408.464,167.914,44.067,158.180
C04760=1029.348,-2.712,408.479,167.912,44.069,158.180
C04761=1029.342,-2.962,408.493,167.909,44.070,158.180
C04762=1029.336,-3.211,408.507,167.907,44.072,158.180
C04763=1029.330,-3.461,408.522,167.905,44.074,158.180
C04764=1029.324,-3.710,408.537,167.902,44.075,158.180
C04765=1029.317,-3.993,408.553,167.899,44.077,158.181
C04766=1029.310,-4.276,408.570,167.896,44.080,158.181
C04767=1029.302,-4.558,408.586,167.893,44.082,158.181
C04768=1029.295,-4.842,408.602,167.891,44.083,158.181
C04769=1029.289,-5.091,408.615,167.888,44.085,158.181
C04770=1029.283,-5.341,408.630,167.885,44.087,158.181
C04771=1029.277,-5.590,408.645,167.883,44.089,158.181
C04772=1029.270,-5.840,408.658,167.880,44.090,158.181
C04773=1029.264,-6.089,408.673,167.877,44.092,158.181
C04774=1029.258,-6.338,408.687,167.875,44.094,158.182
C04775=1029.251,-6.588,408.702,167.872,44.096,158.182
C04776=1029.246,-6.838,408.716,167.869,44.098,158.182
C04777=1029.239,-7.087,408.730,167.867,44.100,158.182
C04778=1029.233,-7.337,408.744,167.864,44.102,158.182
C04779=1029.226,-7.586,408.758,167.861,44.103,158.182
C04780=1029.221,-7.836,408.772,167.860,44.105,158.182
C04781=1029.214,-8.085,408.787,167.857,44.107,158.182
C04782=1029.207,-8.335,408.801,167.855,44.109,158.182
C04783=1029.202,-8.584,408.815,167.852,44.111,158.183
C04784=1029.195,-8.834,408.829,167.849,44.113,158.183
C04785=1029.189,-9.083,408.843,167.847,44.115,158.183
C04786=1029.182,-9.333,408.857,167.844,44.116,158.183
C04787=1029.176,-9.582,408.872,167.841,44.118,158.183
C04788=1029.170,-9.832,408.886,167.839,44.120,158.183
C04789=1029.164,-10.082,408.899,167.836,44.122,158.183
C04790=1029.158,-10.331,408.914,167.833,44.123,158.183
C04791=1029.151,-10.580,408.927,167.831,44.125,158.183
C04792=1029.145,-10.830,408.942,167.828,44.127,158.183
C04793=1029.139,-11.079,408.955,167.825,44.129,158.183
C04794=1029.133,-11.329,408.969,167.824,44.130,158.184
C04795=1029.127,-11.579,408.984,167.821,44.132,158.184
C04796=1029.121,-11.828,408.998,167.819,44.134,158.184
C04797=1029.115,-12.078,409.012,167.816,44.135,158.184
C04798=1029.108,-12.327,409.026,167.813,44.137,158.184
C04799=1029.102,-12.577,409.040,167.811,44.139,158.184
C04800=1029.096,-12.826,409.054,167.808,44.141,158.184
C04801=1029.089,-13.076,409.068,167.805,44.143,158.184
C04802=1029.083,-13.325,409.081,167.802,44.144,158.184
C04803=1029.078,-13.575,409.095,167.800,44.146,158.184
C04804=1029.071,-13.824,409.110,167.797,44.148,158.184
C04805=1029.065,-14.074,409.124,167.795,44.150,158.185
C04806=1029.059,-14.324,409.138,167.792,44.152,158.185
C04807=1029.053,-14.573,409.152,167.789,44.153,158.185
C04808=1029.047,-14.822,409.166,167.788,44.155,158.185
C04809=1029.040,-15.072,409.179,167.785,44.157,158.185
C04810=1029.035,-15.322,409.193,167.782,44.159,158.185
C04811=1029.028,-15.571,409.207,167.780,44.160,158.185
C04812=1029.022,-15.821,409.221,167.777,44.162,158.185
C04813=1029.015,-16.071,409.235,167.774,44.164,158.185
C04814=1029.009,-16.320,409.248,167.772,44.166,158.185
C04815=1029.004,-16.569,409.262,167.769,44.168,158.185
C04816=1028.997,-16.819,409.276,167.767,44.170,158.186
C04817=1028.990,-17.068,409.290,167.764,44.172,158.186
C04818=1028.984,-17.318,409.304,167.761,44.174,158.186
C04819=1028.978,-17.568,409.317,167.759,44.175,158.186
C04820=1028.972,-17.817,409.331,167.756,44.177,158.186
C04821=1028.965,-18.067,409.344,167.753,44.179,158.186
C04822=1028.960,-18.316,409.358,167.751,44.181,158.186
C04823=1028.953,-18.566,409.371,167.748,44.183,158.186
C04824=1028.947,-18.816,409.385,167.745,44.184,158.186
C04825=1028.941,-19.065,409.399,167.743,44.186,158.187
C04826=1028.935,-19.314,409.412,167.740,44.188,158.187
C04827=1028.928,-19.564,409.426,167.738,44.190,158.187
C04828=1028.922,-19.813,409.440,167.735,44.192,158.187
C04829=1028.915,-20.095,409.455,167.731,44.194,158.187
C04830=1028.908,-20.376,409.470,167.729,44.196,158.187
C04831=1028.901,-20.658,409.485,167.726,44.198,158.187
C04832=1028.894,-20.938,409.501,167.722,44.200,158.187
C04833=1028.888,-21.188,409.514,167.720,44.202,158.187
C04834=1028.882,-21.437,409.528,167.717,44.204,158.187
C04835=1028.875,-21.687,409.541,167.715,44.206,158.188
C04836=1028.869,-21.937,409.555,167.712,44.208,158.188
C04837=1028.864,-22.186,409.569,167.709,44.210,158.188
C04838=1028.857,-22.436,409.582,167.707,44.212,158.188
C04839=1028.850,-22.685,409.595,167.704,44.213,158.188
C04840=1028.845,-22.935,409.609,167.701,44.215,158.188
C04841=1028.839,-23.184,409.623,167.699,44.217,158.188
C04842=1028.832,-23.434,409.636,167.696,44.219,158.188
C04843=1028.826,-23.683,409.649,167.694,44.221,158.188
C04844=1028.820,-23.933,409.663,167.691,44.223,158.188
C04845=1028.814,-24.182,409.677,167.688,44.224,158.188
C04846=1028.808,-24.433,409.690,167.685,44.226,158.189
C04847=1028.801,-24.682,409.703,167.683,44.228,158.189
C04848=1028.796,-24.932,409.717,167.680,44.230,158.189
C04849=1028.790,-25.181,409.730,167.678,44.232,158.189
C04850=1028.783,-25.430,409.743,167.675,44.234,158.189
C04851=1028.777,-25.680,409.757,167.672,44.235,158.189
C04852=1028.771,-25.930,409.771,167.670,44.237,158.189
C04853=1028.765,-26.179,409.784,167.667,44.239,158.189
C04854=1028.759,-26.429,409.797,167.664,44.241,158.189
C04855=1028.753,-26.678,409.810,167.662,44.243,158.189
C04856=1028.747,-26.928,409.824,167.659,44.245,158.189
C04857=1028.741,-27.178,409.837,167.656,44.246,158.189
C04858=1028.734,-27.427,409.851,167.654,44.248,158.190
C04859=1028.728,-27.677,409.863,167.651,44.250,158.190
C04860=1028.722,-27.926,409.876,167.648,44.252,158.190
C04861=1028.715,-28.176,409.890,167.646,44.254,158.190
C04862=1028.709,-28.425,409.903,167.643,44.255,158.190
C04863=1028.703,-28.675,409.916,167.641,44.257,158.190
C04864=1028.697,-28.924,409.929,167.638,44.259,158.190
C04865=1028.691,-29.174,409.942,167.635,44.261,158.190
C04866=1028.684,-29.424,409.955,167.633,44.263,158.190
C04867=1028.678,-29.674,409.969,167.630,44.265,158.191
C04868=1028.672,-29.923,409.982,167.628,44.267,158.191
C04869=1028.666,-30.173,409.994,167.624,44.269,158.191
C04870=1028.660,-30.422,410.008,167.621,44.271,158.191
C04871=1028.654,-30.672,410.020,167.619,44.273,158.191
C04872=1028.648,-30.921,410.033,167.616,44.275,158.191
C04873=1028.641,-31.171,410.047,167.614,44.277,158.191
C04874=1028.635,-31.421,410.060,167.611,44.279,158.191
C04875=1028.629,-31.670,410.073,167.608,44.281,158.191
C04876=1028.623,-31.920,410.086,167.606,44.283,158.192
C04877=1028.617,-32.169,410.099,167.603,44.285,158.192
C04878=1028.610,-32.419,410.112,167.600,44.286,158.192
C04879=1028.604,-32.669,410.125,167.598,44.288,158.192
C04880=1028.598,-32.918,410.137,167.595,44.290,158.192
C04881=1028.592,-33.167,410.150,167.592,44.292,158.192
C04882=1028.585,-33.417,410.163,167.590,44.294,158.192
C04883=1028.579,-33.667,410.176,167.586,44.296,158.192
C04884=1028.573,-33.917,410.189,167.584,44.298,158.192
C04885=1028.566,-34.166,410.203,167.581,44.300,158.192
C04886=1028.561,-34.416,410.215,167.578,44.302,158.192
C04887=1028.554,-34.665,410.228,167.576,44.304,158.193
C04888=1028.548,-34.915,410.241,167.573,44.305,158.193
C04889=1028.542,-35.164,410.254,167.571,44.307,158.193
C04890=1028.536,-35.414,410.267,167.568,44.309,158.193
C04891=1028.530,-35.663,410.280,167.565,44.311,158.193
C04892=1028.522,-36.011,410.298,167.562,44.313,158.193
C04893=1028.514,-36.350,410.314,167.557,44.316,158.193
C04894=1028.507,-36.590,410.327,167.554,44.318,158.193
C04895=1028.501,-36.831,410.340,167.552,44.320,158.193
C04896=1028.496,-37.071,410.352,167.550,44.321,158.193
C04897=1028.490,-37.312,410.364,167.548,44.323,158.194
C04898=1028.484,-37.552,410.377,167.545,44.325,158.194
C04899=1028.479,-37.792,410.389,167.542,44.327,158.194
C04900=1028.472,-38.033,410.402,167.540,44.328,158.194
C04901=1028.466,-38.283,410.414,167.537,44.330,158.194
C04902=1028.460,-38.533,410.427,167.534,44.332,158.194
C04903=1028.454,-38.782,410.440,167.531,44.334,158.194
C04904=1028.448,-39.032,410.453,167.528,44.336,158.194
C04905=1028.442,-39.281,410.465,167.526,44.338,158.194
C04906=1028.435,-39.531,410.478,167.523,44.340,158.194
C04907=1028.430,-39.781,410.491,167.520,44.342,158.194
C04908=1028.423,-40.030,410.503,167.518,44.344,158.195
C04909=1028.417,-40.280,410.515,167.515,44.346,158.195
C04910=1028.411,-40.529,410.528,167.511,44.348,158.195
C04911=1028.405,-40.778,410.540,167.509,44.350,158.195
C04912=1028.399,-41.028,410.553,167.506,44.352,158.195
C04913=1028.393,-41.278,410.565,167.504,44.354,158.195
C04914=1028.386,-41.527,410.578,167.501,44.356,158.195
C04915=1028.380,-41.777,410.590,167.498,44.358,158.195
C04916=1028.374,-42.027,410.603,167.496,44.360,158.195
C04917=1028.368,-42.276,410.615,167.492,44.362,158.195
C04918=1028.362,-42.526,410.627,167.490,44.364,158.195
C04919=1028.355,-42.775,410.641,167.487,44.366,158.196
C04920=1028.349,-43.025,410.653,167.484,44.368,158.196
C04921=1028.343,-43.275,410.665,167.482,44.370,158.196
C04922=1028.337,-43.525,410.678,167.479,44.372,158.196
C04923=1028.330,-43.774,410.690,167.477,44.374,158.196
C04924=1028.325,-44.023,410.702,167.473,44.376,158.196
C04925=1028.319,-44.273,410.714,167.470,44.378,158.196
C04926=1028.312,-44.522,410.727,167.468,44.380,158.196
C04927=1028.306,-44.772,410.740,167.465,44.382,158.196
C04928=1028.300,-45.022,410.752,167.462,44.384,158.196
C04929=1028.294,-45.272,410.764,167.460,44.386,158.197
C04930=1028.288,-45.522,410.777,167.457,44.388,158.197
C04931=1028.282,-45.771,410.789,167.454,44.390,158.197
C04932=1028.276,-46.020,410.801,167.451,44.392,158.197
C04933=1028.270,-46.270,410.813,167.448,44.394,158.197
C04934=1028.264,-46.520,410.826,167.446,44.396,158.197
C04935=1028.257,-46.770,410.838,167.443,44.397,158.197
C04936=1028.251,-47.020,410.850,167.441,44.399,158.197
C04937=1028.246,-47.269,410.863,167.438,44.401,158.197
C04938=1028.239,-47.518,410.875,167.434,44.403,158.197
C04939=1028.234,-47.768,410.887,167.432,44.405,158.198
C04940=1028.227,-48.018,410.899,167.429,44.407,158.198
C04941=1028.221,-48.268,410.912,167.427,44.409,158.198
C04942=1028.216,-48.517,410.924,167.424,44.411,158.198
C04943=1028.209,-48.766,410.936,167.421,44.413,158.198
C04944=1028.203,-49.016,410.948,167.418,44.415,158.198
C04945=1028.197,-49.266,410.961,167.415,44.417,158.198
C04946=1028.191,-49.515,410.973,167.412,44.419,158.198
C04947=1028.185,-49.765,410.985,167.410,44.421,158.198
C04948=1028.179,-50.015,410.998,167.407,44.422,158.198
C04949=1028.173,-50.264,411.010,167.404,44.424,158.198
C04950=1028.167,-50.514,411.022,167.402,44.426,158.199
C04951=1028.161,-50.763,411.034,167.398,44.429,158.199
C04952=1028.155,-51.013,411.046,167.396,44.431,158.199
C04953=1028.149,-51.263,411.058,167.393,44.433,158.199
C04954=1028.142,-51.513,411.070,167.391,44.435,158.199
C04955=1028.136,-51.762,411.081,167.387,44.437,158.199
C04956=1028.130,-52.011,411.094,167.384,44.439,158.199
C04957=1028.123,-52.293,411.106,167.381,44.442,158.199
C04958=1028.116,-52.573,411.120,167.378,44.444,158.199
C04959=1028.109,-52.854,411.133,167.375,44.447,158.200
C04960=1028.101,-53.135,411.147,167.371,44.449,158.200
C04961=1028.096,-53.385,411.159,167.369,44.451,158.200
C04962=1028.090,-53.634,411.170,167.366,44.454,158.200
C04963=1028.083,-53.884,411.182,167.364,44.455,158.200
C04964=1028.077,-54.134,411.193,167.360,44.458,158.200
C04965=1028.071,-54.384,411.206,167.358,44.460,158.200
C04966=1028.065,-54.633,411.217,167.355,44.462,158.200
C04967=1028.058,-54.883,411.229,167.353,44.464,158.201
C04968=1028.052,-55.132,411.241,167.349,44.466,158.201
C04969=1028.046,-55.381,411.253,167.346,44.468,158.201
C04970=1028.040,-55.632,411.264,167.344,44.470,158.201
C04971=1028.033,-55.881,411.276,167.341,44.472,158.201
C04972=1028.027,-56.130,411.288,167.337,44.474,158.201
C04973=1028.021,-56.380,411.299,167.335,44.477,158.201
C04974=1028.015,-56.630,411.311,167.332,44.479,158.201
C04975=1028.009,-56.880,411.322,167.330,44.481,158.201
C04976=1028.003,-57.129,411.334,167.326,44.483,158.202
C04977=1027.996,-57.379,411.346,167.324,44.485,158.202
C04978=1027.991,-57.629,411.358,167.321,44.487,158.202
C04979=1027.984,-57.878,411.370,167.318,44.489,158.202
C04980=1027.978,-58.128,411.381,167.315,44.492,158.202
C04981=1027.972,-58.377,411.393,167.312,44.494,158.202
C04982=1027.966,-58.628,411.404,167.310,44.496,158.202
C04983=1027.960,-58.877,411.416,167.307,44.498,158.202
C04984=1027.954,-59.127,411.427,167.304,44.500,158.202
C04985=1027.947,-59.376,411.439,167.301,44.502,158.202
C04986=1027.941,-59.625,411.451,167.298,44.504,158.203
C04987=1027.936,-59.876,411.463,167.296,44.506,158.203
C04988=1027.930,-60.125,411.473,167.292,44.508,158.203
C04989=1027.923,-60.375,411.485,167.290,44.510,158.203
C04990=1027.918,-60.624,411.496,167.287,44.512,158.203
C04991=1027.911,-60.874,411.508,167.285,44.514,158.203
C04992=1027.905,-61.124,411.520,167.281,44.516,158.203
C04993=1027.899,-61.373,411.532,167.278,44.518,158.203
C04994=1027.893,-61.623,411.543,167.276,44.521,158.204
C04995=1027.887,-61.872,411.555,167.272,44.523,158.204
C04996=1027.881,-62.123,411.566,167.270,44.525,158.204
C04997=1027.875,-62.372,411.578,167.267,44.527,158.204
C04998=1027.869,-62.622,411.589,167.264,44.529,158.204
C04999=1027.863,-62.871,411.600,167.261,44.531,158.204
C05000=1027.857,-63.121,411.612,167.258,44.533,158.204
C05001=1027.851,-63.370,411.623,167.256,44.535,158.204
C05002=1027.845,-63.620,411.635,167.253,44.537,158.204
C05003=1027.839,-63.870,411.646,167.250,44.540,158.204
C05004=1027.833,-64.120,411.658,167.247,44.542,158.205
C05005=1027.827,-64.369,411.669,167.244,44.544,158.205
C05006=1027.821,-64.619,411.680,167.242,44.546,158.205
C05007=1027.816,-64.869,411.692,167.238,44.548,158.205
C05008=1027.809,-65.118,411.704,167.236,44.550,158.205
C05009=1027.803,-65.368,411.715,167.233,44.552,158.205
C05010=1027.797,-65.618,411.726,167.230,44.554,158.205
C05011=1027.791,-65.867,411.738,167.227,44.556,158.205
C05012=1027.785,-66.116,411.748,167.224,44.558,158.205
C05013=1027.779,-66.367,411.760,167.222,44.561,158.205
C05014=1027.774,-66.616,411.771,167.219,44.563,158.206
C05015=1027.767,-66.866,411.783,167.216,44.565,158.206
C05016=1027.761,-67.116,411.794,167.213,44.567,158.206
C05017=1027.755,-67.366,411.805,167.210,44.569,158.206
C05018=1027.749,-67.615,411.817,167.207,44.571,158.206
C05019=1027.744,-67.864,411.828,167.204,44.573,158.206
C05020=1027.738,-68.115,411.840,167.201,44.575,158.206
C05021=1027.731,-68.396,411.852,167.198,44.577,158.206
C05022=1027.725,-68.678,411.864,167.195,44.580,158.206
C05023=1027.717,-68.960,411.878,167.192,44.582,158.206
C05024=1027.711,-69.242,411.890,167.188,44.585,158.206
C05025=1027.704,-69.492,411.901,167.186,44.587,158.207
C05026=1027.699,-69.742,411.913,167.183,44.589,158.207
C05027=1027.694,-69.991,411.924,167.180,44.591,158.207
C05028=1027.687,-70.241,411.936,167.177,44.593,158.207
C05029=1027.681,-70.490,411.946,167.174,44.595,158.207
C05030=1027.675,-70.740,411.957,167.172,44.597,158.207
C05031=1027.669,-70.990,411.969,167.168,44.599,158.207
C05032=1027.663,-71.240,411.979,167.166,44.601,158.207
C05033=1027.658,-71.489,411.991,167.163,44.603,158.207
C05034=1027.652,-71.740,412.002,167.160,44.605,158.207
C05035=1027.646,-71.988,412.014,167.157,44.607,158.207
C05036=1027.640,-72.238,412.025,167.154,44.609,158.207
C05037=1027.634,-72.487,412.035,167.152,44.611,158.208
C05038=1027.628,-72.738,412.047,167.149,44.613,158.208
C05039=1027.622,-72.987,412.058,167.145,44.615,158.208
C05040=1027.617,-73.237,412.069,167.143,44.617,158.208
C05041=1027.611,-73.487,412.080,167.140,44.620,158.208
C05042=1027.605,-73.737,412.091,167.137,44.622,158.208
C05043=1027.600,-73.986,412.102,167.134,44.624,158.208
C05044=1027.594,-74.236,412.113,167.132,44.626,158.208
C05045=1027.587,-74.486,412.124,167.129,44.628,158.208
C05046=1027.582,-74.735,412.135,167.125,44.630,158.208
C05047=1027.576,-74.985,412.146,167.123,44.632,158.208
C05048=1027.569,-75.235,412.157,167.120,44.634,158.209
C05049=1027.563,-75.485,412.167,167.117,44.637,158.209
C05050=1027.558,-75.734,412.178,167.114,44.639,158.209
C05051=1027.552,-75.984,412.188,167.111,44.641,158.209
C05052=1027.546,-76.234,412.200,167.108,44.643,158.209
C05053=1027.540,-76.483,412.211,167.105,44.645,158.209
C05054=1027.534,-76.733,412.221,167.103,44.647,158.209
C05055=1027.528,-76.982,412.232,167.099,44.650,158.209
C05056=1027.522,-77.232,412.243,167.097,44.651,158.209
C05057=1027.516,-77.482,412.253,167.093,44.654,158.210
C05058=1027.510,-77.732,412.264,167.091,44.656,158.210
C05059=1027.504,-77.981,412.275,167.088,44.658,158.210
C05060=1027.499,-78.231,412.286,167.084,44.660,158.210
C05061=1027.492,-78.481,412.296,167.082,44.663,158.210
C05062=1027.486,-78.731,412.307,167.079,44.665,158.210
C05063=1027.480,-78.980,412.317,167.076,44.667,158.210
C05064=1027.475,-79.230,412.328,167.073,44.669,158.210
C05065=1027.469,-79.479,412.339,167.071,44.671,158.210
C05066=1027.464,-79.729,412.349,167.067,44.674,158.211
C05067=1027.456,-79.979,412.360,167.065,44.676,158.211
C05068=1027.451,-80.229,412.371,167.062,44.678,158.211
C05069=1027.445,-80.479,412.381,167.059,44.681,158.211
C05070=1027.439,-80.728,412.391,167.056,44.683,158.211
C05071=1027.433,-80.978,412.402,167.052,44.685,158.211
C05072=1027.426,-81.228,412.412,167.050,44.688,158.211
C05073=1027.421,-81.478,412.423,167.047,44.690,158.211
C05074=1027.414,-81.727,412.433,167.044,44.693,158.212
C05075=1027.409,-81.977,412.444,167.041,44.695,158.212
C05076=1027.403,-82.226,412.454,167.038,44.697,158.212
C05077=1027.397,-82.476,412.464,167.035,44.699,158.212
C05078=1027.391,-82.726,412.475,167.033,44.701,158.212
C05079=1027.384,-82.976,412.485,167.029,44.704,158.212
C05080=1027.378,-83.226,412.496,167.027,44.706,158.212
C05081=1027.372,-83.475,412.506,167.023,44.708,158.212
C05082=1027.367,-83.725,412.516,167.021,44.711,158.213
C05083=1027.361,-83.974,412.527,167.018,44.713,158.213
C05084=1027.355,-84.224,412.537,167.015,44.715,158.213
C05085=1027.348,-84.509,412.548,167.011,44.718,158.213
C05086=1027.341,-84.792,412.560,167.008,44.721,158.213
C05087=1027.334,-85.076,412.572,167.004,44.724,158.213
C05088=1027.327,-85.361,412.584,167.002,44.726,158.213
C05089=1027.321,-85.611,412.594,166.998,44.729,158.213
C05090=1027.315,-85.860,412.604,166.996,44.731,158.214
C05091=1027.309,-86.110,412.614,166.992,44.733,158.214
C05092=1027.303,-86.360,412.625,166.990,44.735,158.214
C05093=1027.297,-86.609,412.634,166.987,44.737,158.214
C05094=1027.292,-86.859,412.645,166.984,44.740,158.214
C05095=1027.286,-87.109,412.656,166.981,44.742,158.214
C05096=1027.280,-87.358,412.666,166.978,44.744,158.214
C05097=1027.274,-87.608,412.676,166.975,44.747,158.214
C05098=1027.268,-87.858,412.686,166.973,44.749,158.215
C05099=1027.262,-88.108,412.696,166.969,44.751,158.215
C05100=1027.256,-88.357,412.706,166.967,44.754,158.215
C05101=1027.250,-88.607,412.717,166.963,44.756,158.215
C05102=1027.244,-88.857,412.726,166.960,44.758,158.215
C05103=1027.239,-89.107,412.737,166.957,44.761,158.215
C05104=1027.232,-89.356,412.747,166.954,44.763,158.215
C05105=1027.227,-89.606,412.757,166.952,44.765,158.215
C05106=1027.221,-89.856,412.767,166.948,44.768,158.215
C05107=1027.215,-90.105,412.777,166.946,44.770,158.216
C05108=1027.209,-90.355,412.787,166.942,44.772,158.216
C05109=1027.203,-90.605,412.797,166.940,44.775,158.216
C05110=1027.197,-90.854,412.807,166.937,44.777,158.216
C05111=1027.192,-91.104,412.817,166.934,44.779,158.216
C05112=1027.186,-91.354,412.827,166.931,44.782,158.216
C05113=1027.180,-91.603,412.838,166.928,44.784,158.216
C05114=1027.174,-91.853,412.847,166.925,44.786,158.216
C05115=1027.169,-92.103,412.857,166.923,44.788,158.216
C05116=1027.162,-92.353,412.867,166.919,44.791,158.217
C05117=1027.157,-92.602,412.878,166.916,44.793,158.217
C05118=1027.150,-92.852,412.887,166.913,44.795,158.217
C05119=1027.145,-93.102,412.898,166.910,44.797,158.217
C05120=1027.139,-93.352,412.907,166.908,44.799,158.217
C05121=1027.134,-93.602,412.917,166.904,44.802,158.217
C05122=1027.128,-93.851,412.927,166.902,44.804,158.217
C05123=1027.122,-94.101,412.937,166.898,44.806,158.217
C05124=1027.116,-94.351,412.947,166.896,44.809,158.217
C05125=1027.111,-94.601,412.957,166.893,44.811,158.218
C05126=1027.104,-94.851,412.967,166.890,44.813,158.218
C05127=1027.099,-95.099,412.977,166.887,44.816,158.218
C05128=1027.093,-95.349,412.987,166.884,44.818,158.218
C05129=1027.088,-95.599,412.997,166.881,44.820,158.218
C05130=1027.081,-95.849,413.007,166.879,44.823,158.218
C05131=1027.076,-96.099,413.017,166.875,44.825,158.218
C05132=1027.070,-96.349,413.026,166.872,44.827,158.218
C05133=1027.065,-96.598,413.036,166.869,44.830,158.218
C05134=1027.059,-96.848,413.046,166.866,44.832,158.219
C05135=1027.053,-97.098,413.057,166.864,44.834,158.219
C05136=1027.047,-97.347,413.066,166.860,44.837,158.219
C05137=1027.041,-97.598,413.076,166.858,44.839,158.219
C05138=1027.036,-97.847,413.085,166.854,44.842,158.219
C05139=1027.030,-98.096,413.095,166.852,44.844,158.219
C05140=1027.024,-98.346,413.105,166.848,44.846,158.219
C05141=1027.017,-98.596,413.114,166.846,44.848,158.219
C05142=1027.013,-98.845,413.124,166.842,44.851,158.220
C05143=1027.006,-99.095,413.133,166.840,44.853,158.220
C05144=1027.001,-99.346,413.142,166.836,44.856,158.220
C05145=1026.994,-99.595,413.152,166.834,44.858,158.220
C05146=1026.989,-99.846,413.162,166.830,44.861,158.220
C05147=1026.983,-100.095,413.171,166.828,44.863,158.220
C05148=1026.977,-100.344,413.181,166.826,44.866,158.220
C05149=1026.970,-100.631,413.192,166.822,44.868,158.220
C05150=1026.963,-100.917,413.203,166.819,44.871,158.221
C05151=1026.957,-101.203,413.214,166.815,44.874,158.221
C05152=1026.951,-101.490,413.225,166.812,44.877,158.221
C05153=1026.944,-101.739,413.234,166.808,44.879,158.221
C05154=1026.938,-101.989,413.244,166.806,44.882,158.221
C05155=1026.933,-102.239,413.252,166.802,44.884,158.221
C05156=1026.928,-102.489,413.262,166.800,44.886,158.221
C05157=1026.921,-102.739,413.272,166.796,44.889,158.221
C05158=1026.916,-102.988,413.281,166.794,44.891,158.222
C05159=1026.910,-103.238,413.291,166.790,44.893,158.222
C05160=1026.903,-103.487,413.300,166.788,44.896,158.222
C05161=1026.898,-103.737,413.309,166.784,44.898,158.222
C05162=1026.893,-103.987,413.319,166.782,44.901,158.222
C05163=1026.887,-104.237,413.329,166.778,44.903,158.222
C05164=1026.881,-104.486,413.338,166.776,44.906,158.222
C05165=1026.875,-104.737,413.347,166.773,44.908,158.222
C05166=1026.869,-104.986,413.356,166.770,44.911,158.223
C05167=1026.863,-105.235,413.365,166.767,44.913,158.223
C05168=1026.858,-105.486,413.376,166.764,44.916,158.223
C05169=1026.852,-105.736,413.384,166.761,44.918,158.223
C05170=1026.847,-105.985,413.394,166.758,44.921,158.223
C05171=1026.840,-106.235,413.403,166.755,44.923,158.223
C05172=1026.835,-106.485,413.412,166.752,44.926,158.223
C05173=1026.829,-106.734,413.421,166.749,44.928,158.224
C05174=1026.823,-106.984,413.431,166.746,44.930,158.224
C05175=1026.818,-107.234,413.439,166.744,44.933,158.224
C05176=1026.811,-107.484,413.449,166.740,44.935,158.224
C05177=1026.806,-107.733,413.458,166.738,44.938,158.224
C05178=1026.800,-107.983,413.467,166.734,44.940,158.224
C05179=1026.794,-108.233,413.476,166.732,44.943,158.224
C05180=1026.788,-108.483,413.485,166.728,44.946,158.224
C05181=1026.782,-108.733,413.495,166.726,44.948,158.225
C05182=1026.777,-108.982,413.503,166.722,44.951,158.225
C05183=1026.771,-109.232,413.513,166.720,44.953,158.225
C05184=1026.765,-109.481,413.522,166.716,44.956,158.225
C05185=1026.759,-109.732,413.531,166.714,44.958,158.225
C05186=1026.754,-109.981,413.540,166.710,44.960,158.225
C05187=1026.748,-110.231,413.549,166.708,44.963,158.225
C05188=1026.742,-110.481,413.558,166.704,44.965,158.225
C05189=1026.737,-110.731,413.567,166.702,44.968,158.226
C05190=1026.730,-110.980,413.576,166.698,44.971,158.226
C05191=1026.725,-111.230,413.585,166.696,44.973,158.226
C05192=1026.719,-111.480,413.594,166.692,44.976,158.226
C05193=1026.714,-111.730,413.603,166.690,44.978,158.226
C05194=1026.708,-111.980,413.612,166.686,44.981,158.226
C05195=1026.702,-112.229,413.621,166.684,44.983,158.227
C05196=1026.696,-112.480,413.630,166.681,44.986,158.227
C05197=1026.691,-112.729,413.639,166.678,44.988,158.227
C05198=1026.685,-112.979,413.648,166.675,44.991,158.227
C05199=1026.679,-113.228,413.657,166.672,44.993,158.227
C05200=1026.674,-113.478,413.665,166.669,44.996,158.227
C05201=1026.668,-113.728,413.674,166.666,44.998,158.227
C05202=1026.663,-113.977,413.684,166.663,45.001,158.227
C05203=1026.657,-114.228,413.692,166.660,45.003,158.227
C05204=1026.651,-114.477,413.700,166.657,45.006,158.228
C05205=1026.645,-114.727,413.710,166.654,45.009,158.228
C05206=1026.639,-114.977,413.718,166.651,45.011,158.228
C05207=1026.634,-115.227,413.727,166.647,45.014,158.228
C05208=1026.628,-115.476,413.736,166.645,45.017,158.228
C05209=1026.623,-115.726,413.745,166.641,45.019,158.228
C05210=1026.616,-115.976,413.753,166.639,45.021,158.228
C05211=1026.611,-116.225,413.762,166.636,45.024,158.229
C05212=1026.605,-116.476,413.771,166.633,45.026,158.229
C05213=1026.598,-116.761,413.781,166.630,45.029,158.229
C05214=1026.592,-117.048,413.791,166.626,45.032,158.229
C05215=1026.585,-117.333,413.801,166.623,45.036,158.229
C05216=1026.579,-117.619,413.811,166.620,45.039,158.229
C05217=1026.573,-117.869,413.819,166.616,45.041,158.230
C05218=1026.567,-118.119,413.828,166.614,45.044,158.230
C05219=1026.562,-118.369,413.836,166.610,45.047,158.230
C05220=1026.556,-118.618,413.846,166.608,45.049,158.230
C05221=1026.550,-118.868,413.854,166.604,45.051,158.230
C05222=1026.544,-119.118,413.862,166.601,45.054,158.230
C05223=1026.539,-119.367,413.871,166.599,45.057,158.230
C05224=1026.533,-119.618,413.880,166.595,45.059,158.230
C05225=1026.527,-119.867,413.888,166.593,45.062,158.231
C05226=1026.522,-120.117,413.896,166.589,45.065,158.231
C05227=1026.516,-120.367,413.906,166.587,45.067,158.231
C05228=1026.511,-120.616,413.914,166.583,45.070,158.231
C05229=1026.505,-120.866,413.922,166.581,45.073,158.231
C05230=1026.499,-121.116,413.931,166.577,45.075,158.231
C05231=1026.493,-121.366,413.939,166.575,45.077,158.232
C05232=1026.488,-121.616,413.948,166.572,45.080,158.232
C05233=1026.482,-121.866,413.956,166.569,45.083,158.232
C05234=1026.476,-122.115,413.965,166.566,45.085,158.232
C05235=1026.471,-122.365,413.973,166.563,45.088,158.232
C05236=1026.466,-122.615,413.982,166.560,45.091,158.232
C05237=1026.459,-122.865,413.990,166.556,45.093,158.232
C05238=1026.454,-123.115,413.998,166.554,45.096,158.233
C05239=1026.449,-123.364,414.007,166.551,45.099,158.233
C05240=1026.443,-123.614,414.015,166.548,45.101,158.233
C05241=1026.437,-123.864,414.024,166.545,45.104,158.233
C05242=1026.432,-124.114,414.032,166.542,45.106,158.233
C05243=1026.426,-124.363,414.040,166.539,45.109,158.233
C05244=1026.420,-124.613,414.048,166.537,45.112,158.234
C05245=1026.414,-124.863,414.057,166.533,45.114,158.234
C05246=1026.408,-125.113,414.065,166.531,45.117,158.234
C05247=1026.403,-125.363,414.074,166.527,45.120,158.234
C05248=1026.397,-125.612,414.082,166.524,45.123,158.234
C05249=1026.392,-125.862,414.090,166.521,45.126,158.234
C05250=1026.385,-126.112,414.098,166.518,45.128,158.234
C05251=1026.380,-126.362,414.106,166.515,45.130,158.234
C05252=1026.375,-126.612,414.115,166.512,45.133,158.235
C05253=1026.369,-126.861,414.122,166.510,45.136,158.235
C05254=1026.364,-127.111,414.131,166.506,45.139,158.235
C05255=1026.357,-127.361,414.139,166.503,45.141,158.235
C05256=1026.352,-127.611,414.148,166.500,45.144,158.235
C05257=1026.346,-127.860,414.156,166.497,45.147,158.235
C05258=1026.341,-128.109,414.164,166.494,45.149,158.235
C05259=1026.337,-128.359,414.173,166.492,45.151,158.236
C05260=1026.332,-128.609,414.183,166.489,45.152,158.235
C05261=1026.329,-128.859,414.193,166.486,45.154,158.235
C05262=1026.326,-129.109,414.203,166.484,45.154,158.235
C05263=1026.322,-129.358,414.215,166.481,45.154,158.235
C05264=1026.321,-129.608,414.227,166.478,45.154,158.235
C05265=1026.320,-129.857,414.239,166.476,45.153,158.234
C05266=1026.319,-130.107,414.253,166.474,45.151,158.234
C05267=1026.319,-130.357,414.266,166.472,45.150,158.233
C05268=1026.319,-130.607,414.281,166.470,45.147,158.233
C05269=1026.320,-130.857,414.296,166.468,45.144,158.232
C05270=1026.321,-131.107,414.311,166.466,45.141,158.231
C05271=1026.323,-131.356,414.327,166.464,45.138,158.231
C05272=1026.326,-131.606,414.344,166.462,45.133,158.230
C05273=1026.329,-131.857,414.360,166.461,45.128,158.229
C05274=1026.332,-132.106,414.378,166.459,45.123,158.228
C05275=1026.337,-132.356,414.396,166.458,45.117,158.226
C05276=1026.341,-132.606,414.416,166.456,45.111,158.225
C05277=1026.037,-132.631,414.092,166.409,45.374,158.264
C05278=1026.031,-132.382,414.074,166.410,45.380,158.266
C05279=1026.027,-132.132,414.055,166.411,45.386,158.267
C05280=1026.024,-131.882,414.037,166.413,45.391,158.268
C05281=1026.021,-131.633,414.020,166.414,45.396,158.269
C05282=1026.018,-131.383,414.003,166.416,45.400,158.270
C05283=1026.016,-131.132,413.987,166.418,45.404,158.270
C05284=1026.015,-130.882,413.972,166.419,45.407,158.271
C05285=1026.014,-130.632,413.957,166.422,45.410,158.272
C05286=1026.013,-130.383,413.943,166.424,45.412,158.272
C05287=1026.013,-130.133,413.929,166.426,45.414,158.273
C05288=1026.014,-129.884,413.916,166.428,45.416,158.273
C05289=1026.016,-129.634,413.903,166.431,45.417,158.274
C05290=1026.018,-129.384,413.891,166.433,45.417,158.274
C05291=1026.020,-129.134,413.880,166.435,45.417,158.274
C05292=1026.023,-128.884,413.869,166.438,45.416,158.275
C05293=1026.026,-128.635,413.859,166.441,45.415,158.275
C05294=1026.031,-128.385,413.849,166.444,45.414,158.275
C05295=1026.036,-128.135,413.840,166.447,45.412,158.275
C05296=1026.041,-127.886,413.832,166.449,45.409,158.275
C05297=1026.046,-127.636,413.823,166.452,45.406,158.274
C05298=1026.052,-127.387,413.815,166.455,45.404,158.274
C05299=1026.058,-127.137,413.807,166.458,45.401,158.274
C05300=1026.064,-126.888,413.799,166.462,45.398,158.274
C05301=1026.069,-126.637,413.791,166.464,45.396,158.274
C05302=1026.075,-126.388,413.783,166.467,45.393,158.274
C05303=1026.080,-126.137,413.774,166.470,45.390,158.273
C05304=1026.086,-125.888,413.766,166.473,45.388,158.273
C05305=1026.092,-125.638,413.758,166.477,45.385,158.273
C05306=1026.097,-125.389,413.749,166.479,45.382,158.273
C05307=1026.103,-125.139,413.742,166.482,45.379,158.273
C05308=1026.109,-124.888,413.733,166.485,45.376,158.273
C05309=1026.115,-124.639,413.726,166.488,45.373,158.273
C05310=1026.120,-124.389,413.717,166.491,45.370,158.272
C05311=1026.125,-124.139,413.709,166.494,45.368,158.272
C05312=1026.132,-123.889,413.700,166.497,45.365,158.272
C05313=1026.137,-123.639,413.692,166.500,45.363,158.272
C05314=1026.142,-123.390,413.683,166.503,45.360,158.272
C05315=1026.147,-123.140,413.675,166.506,45.358,158.272
C05316=1026.154,-122.890,413.667,166.509,45.355,158.272
C05317=1026.159,-122.640,413.658,166.512,45.352,158.271
C05318=1026.165,-122.390,413.650,166.515,45.349,158.271
C05319=1026.171,-122.141,413.642,166.518,45.346,158.271
C05320=1026.176,-121.891,413.633,166.521,45.344,158.271
C05321=1026.182,-121.641,413.624,166.524,45.341,158.271
C05322=1026.187,-121.391,413.616,166.526,45.339,158.271
C05323=1026.193,-121.142,413.608,166.530,45.336,158.271
C05324=1026.199,-120.891,413.599,166.533,45.333,158.270
C05325=1026.204,-120.642,413.591,166.536,45.331,158.270
C05326=1026.210,-120.393,413.581,166.539,45.328,158.270
C05327=1026.216,-120.142,413.573,166.541,45.325,158.270
C05328=1026.222,-119.893,413.565,166.545,45.323,158.270
C05329=1026.227,-119.643,413.556,166.547,45.320,158.270
C05330=1026.232,-119.393,413.548,166.551,45.317,158.270
C05331=1026.239,-119.143,413.540,166.554,45.314,158.269
C05332=1026.244,-118.894,413.531,166.557,45.312,158.269
C05333=1026.249,-118.644,413.523,166.560,45.309,158.269
C05334=1026.255,-118.394,413.513,166.562,45.306,158.269
C05335=1026.261,-118.145,413.505,166.566,45.303,158.269
C05336=1026.267,-117.894,413.496,166.568,45.301,158.269
C05337=1026.273,-117.644,413.488,166.572,45.299,158.269
C05338=1026.279,-117.359,413.478,166.575,45.296,158.268
C05339=1026.286,-117.073,413.467,166.578,45.292,158.268
C05340=1026.292,-116.787,413.458,166.582,45.289,158.268
C05341=1026.299,-116.501,413.448,166.585,45.286,158.268
C05342=1026.304,-116.251,413.440,166.589,45.284,158.268
C05343=1026.310,-116.002,413.430,166.591,45.281,158.268
C05344=1026.316,-115.752,413.422,166.594,45.278,158.267
C05345=1026.321,-115.502,413.413,166.597,45.275,158.267
C05346=1026.327,-115.252,413.405,166.600,45.273,158.267
C05347=1026.333,-115.003,413.396,166.604,45.270,158.267
C05348=1026.339,-114.753,413.387,166.606,45.268,158.267
C05349=1026.344,-114.503,413.378,166.609,45.265,158.267
C05350=1026.350,-114.253,413.369,166.612,45.263,158.267
C05351=1026.356,-114.003,413.360,166.615,45.260,158.266
C05352=1026.361,-113.754,413.352,166.618,45.257,158.266
C05353=1026.367,-113.504,413.342,166.621,45.255,158.266
C05354=1026.372,-113.254,413.334,166.624,45.252,158.266
C05355=1026.378,-113.004,413.325,166.627,45.249,158.266
C05356=1026.384,-112.755,413.316,166.630,45.247,158.266
C05357=1026.390,-112.505,413.308,166.633,45.244,158.266
C05358=1026.396,-112.255,413.298,166.636,45.241,158.265
C05359=1026.402,-112.005,413.289,166.639,45.239,158.265
C05360=1026.407,-111.755,413.281,166.642,45.236,158.265
C05361=1026.413,-111.506,413.271,166.645,45.234,158.265
C05362=1026.418,-111.256,413.263,166.648,45.231,158.265
C05363=1026.425,-111.006,413.253,166.651,45.229,158.265
C05364=1026.430,-110.756,413.245,166.654,45.226,158.265
C05365=1026.436,-110.507,413.235,166.657,45.224,158.265
C05366=1026.441,-110.257,413.227,166.660,45.221,158.264
C05367=1026.448,-110.007,413.217,166.663,45.219,158.264
C05368=1026.453,-109.757,413.209,166.666,45.216,158.264
C05369=1026.459,-109.507,413.199,166.669,45.213,158.264
C05370=1026.464,-109.258,413.191,166.672,45.211,158.264
C05371=1026.470,-109.008,413.181,166.675,45.208,158.264
C05372=1026.476,-108.758,413.173,166.678,45.205,158.264
C05373=1026.482,-108.508,413.163,166.681,45.203,158.264
C05374=1026.487,-108.259,413.155,166.684,45.200,158.263
C05375=1026.493,-108.009,413.145,166.687,45.197,158.263
C05376=1026.499,-107.759,413.135,166.689,45.195,158.263
C05377=1026.505,-107.509,413.127,166.693,45.192,158.263
C05378=1026.511,-107.260,413.117,166.695,45.190,158.263
C05379=1026.516,-107.010,413.109,166.699,45.187,158.263
C05380=1026.522,-106.760,413.099,166.701,45.185,158.262
C05381=1026.528,-106.511,413.090,166.705,45.183,158.262
C05382=1026.534,-106.261,413.081,166.707,45.180,158.262
C05383=1026.540,-106.011,413.072,166.711,45.177,158.262
C05384=1026.545,-105.761,413.062,166.713,45.175,158.262
C05385=1026.551,-105.511,413.053,166.716,45.172,158.262
C05386=1026.557,-105.261,413.044,166.719,45.170,158.262
C05387=1026.562,-105.012,413.034,166.722,45.167,158.262
C05388=1026.569,-104.762,413.025,166.726,45.165,158.262
C05389=1026.574,-104.513,413.016,166.728,45.162,158.261
C05390=1026.580,-104.263,413.007,166.732,45.159,158.261
C05391=1026.585,-104.013,412.997,166.734,45.157,158.261
C05392=1026.591,-103.763,412.988,166.738,45.154,158.261
C05393=1026.597,-103.513,412.979,166.740,45.152,158.261
C05394=1026.603,-103.263,412.969,166.744,45.149,158.261
C05395=1026.609,-103.014,412.960,166.746,45.147,158.261
C05396=1026.615,-102.764,412.950,166.750,45.144,158.260
C05397=1026.620,-102.514,412.941,166.752,45.142,158.260
C05398=1026.625,-102.265,412.932,166.756,45.139,158.260
C05399=1026.632,-102.015,412.922,166.758,45.137,158.260
C05400=1026.638,-101.765,412.912,166.762,45.135,158.260
C05401=1026.643,-101.516,412.903,166.764,45.132,158.260
C05402=1026.650,-101.229,412.892,166.767,45.129,158.260
C05403=1026.657,-100.943,412.881,166.771,45.126,158.259
C05404=1026.664,-100.656,412.871,166.774,45.123,158.259
C05405=1026.670,-100.371,412.859,166.778,45.121,158.259
C05406=1026.676,-100.120,412.851,166.781,45.118,158.259
C05407=1026.681,-99.870,412.840,166.783,45.115,158.259
C05408=1026.687,-99.621,412.831,166.787,45.113,158.259
C05409=1026.693,-99.371,412.822,166.789,45.110,158.259
C05410=1026.699,-99.122,412.812,166.793,45.108,158.259
C05411=1026.705,-98.872,412.802,166.795,45.105,158.258
C05412=1026.711,-98.622,412.792,166.799,45.103,158.258
C05413=1026.716,-98.373,412.783,166.801,45.101,158.258
C05414=1026.722,-98.123,412.774,166.805,45.098,158.258
C05415=1026.729,-97.873,412.764,166.807,45.096,158.258
C05416=1026.735,-97.623,412.754,166.811,45.093,158.258
C05417=1026.740,-97.374,412.745,166.813,45.091,158.258
C05418=1026.746,-97.124,412.735,166.817,45.088,158.258
C05419=1026.751,-96.874,412.725,166.819,45.086,158.257
C05420=1026.757,-96.624,412.715,166.822,45.084,158.257
C05421=1026.763,-96.374,412.705,166.825,45.081,158.257
C05422=1026.768,-96.125,412.696,166.828,45.079,158.257
C05423=1026.774,-95.875,412.686,166.831,45.077,158.257
C05424=1026.780,-95.625,412.676,166.834,45.074,158.257
C05425=1026.786,-95.376,412.665,166.837,45.072,158.257
C05426=1026.792,-95.126,412.656,166.840,45.069,158.257
C05427=1026.797,-94.876,412.646,166.843,45.067,158.257
C05428=1026.803,-94.627,412.636,166.846,45.065,158.257
C05429=1026.808,-94.376,412.626,166.848,45.062,158.256
C05430=1026.815,-94.127,412.617,166.852,45.060,158.256
C05431=1026.820,-93.876,412.607,166.854,45.058,158.256
C05432=1026.826,-93.627,412.596,166.858,45.055,158.256
C05433=1026.831,-93.378,412.586,166.860,45.053,158.256
C05434=1026.837,-93.128,412.577,166.864,45.050,158.256
C05435=1026.843,-92.878,412.567,166.866,45.048,158.256
C05436=1026.849,-92.628,412.557,166.869,45.046,158.256
C05437=1026.855,-92.379,412.546,166.872,45.043,158.255
C05438=1026.861,-92.129,412.537,166.875,45.041,158.255
C05439=1026.866,-91.879,412.527,166.878,45.038,158.255
C05440=1026.873,-91.629,412.517,166.881,45.036,158.255
C05441=1026.878,-91.380,412.506,166.884,45.033,158.255
C05442=1026.884,-91.130,412.497,166.887,45.031,158.255
C05443=1026.889,-90.880,412.487,166.891,45.029,158.255
C05444=1026.896,-90.631,412.476,166.893,45.026,158.255
C05445=1026.901,-90.381,412.466,166.895,45.024,158.255
C05446=1026.907,-90.131,412.457,166.899,45.022,158.254
C05447=1026.913,-89.881,412.447,166.901,45.020,158.254
C05448=1026.919,-89.632,412.436,166.905,45.017,158.254
C05449=1026.925,-89.382,412.426,166.907,45.015,158.254
C05450=1026.931,-89.132,412.417,166.911,45.012,158.254
C05451=1026.937,-88.883,412.406,166.913,45.010,158.254
C05452=1026.943,-88.633,412.396,166.917,45.008,158.254
C05453=1026.948,-88.383,412.386,166.919,45.005,158.254
C05454=1026.955,-88.133,412.376,166.922,45.003,158.253
C05455=1026.960,-87.883,412.366,166.926,45.001,158.253
C05456=1026.967,-87.634,412.355,166.928,44.998,158.253
C05457=1026.972,-87.384,412.345,166.932,44.996,158.253
